 fbDosingStChart2(
	bWrite:= VIS.bDispencer1Dose, 
	udiCycleTime:= 5,
	lrAiData0:= VIS.lrDispencer2ActPos,
	lrAiData1:= VIS.lrDispencer12LifterActPos, 
	lrAiData2:= BOOL_TO_LREAL(P02_Dispencers.QbDispencer2SuckingValveActuator),
	lrAiData3:= BOOL_TO_LREAL(P02_Dispencers.QbDispencer2DosingValveActuator), 
	lrAiData4:= BOOL_TO_LREAL(P02_Dispencers.QbDispencer2DropCatcherValveActuator), 
	AiData=> VIS.AStAsChartDose2[0] );
	
fbDosingChart3(
	bWrite:= VIS.bDispencer3Dose, 
	nCycleTime:= 5,//nChartCycleTime, 
	lrData1:= VIS.lrDispencer3ActPos, 
	lrData2:= VIS.lrDispencer34LifterActPos, 
	bData3:= P02_Dispencers.QbDispencer3SuckingValveActuator, 
	bData4:= P02_Dispencers.QbDispencer3DosingValveActuator,
	bData5:= P02_Dispencers.QbDispencer3DropCatcherValveActuator,
	AsData=>VIS.AsChartDose3 );
	
 fbDosingStChart3(
	bWrite:= VIS.bDispencer1Dose, 
	udiCycleTime:= 5,
	lrAiData0:= VIS.lrDispencer3ActPos,
	lrAiData1:= VIS.lrDispencer34LifterActPos, 
	lrAiData2:= BOOL_TO_LREAL(P02_Dispencers.QbDispencer3SuckingValveActuator),
	lrAiData3:= BOOL_TO_LREAL(P02_Dispencers.QbDispencer3DosingValveActuator), 
	lrAiData4:= BOOL_TO_LREAL(P02_Dispencers.QbDispencer3DropCatcherValveActuator), 
	AiData=> VIS.AStAsChartDose3[0] );

fbDosingChart4(
	bWrite:= VIS.bDispencer4Dose, 
	nCycleTime:= 5,//nChartCycleTime, 
	lrData1:= VIS.lrDispencer4ActPos, 
	lrData2:= VIS.lrDispencer34LifterActPos, 
	bData3:= P02_Dispencers.QbDispencer4SuckingValveActuator, 
	bData4:= P02_Dispencers.QbDispencer4DosingValveActuator,
	bData5:= P02_Dispencers.QbDispencer4DropCatcherValveActuator,
	AsData=>VIS.AsChartDose4 );

fbDosingStChart4(
	bWrite:= VIS.bDispencer1Dose, 
	udiCycleTime:= 5,
	lrAiData0:= VIS.lrDispencer4ActPos,
	lrAiData1:= VIS.lrDispencer34LifterActPos, 
	lrAiData2:= BOOL_TO_LREAL(P02_Dispencers.QbDispencer4SuckingValveActuator),
	lrAiData3:= BOOL_TO_LREAL(P02_Dispencers.QbDispencer4DosingValveActuator), 
	lrAiData4:= BOOL_TO_LREAL(P02_Dispencers.QbDispencer4DropCatcherValveActuator), 
	AiData=> VIS.AStAsChartDose4[0] );
END_ACTION

ACTION aDropCatcher:
(**Uruchamianie ssawki tacek**)
P02_Dispencers.QbDispencerDropCatcherSuck;
IF (P00_PackML.fbPMLAuto.ePMLState = E_PMLState.ePMLState_EXECUTE OR P00_PackML.fbPMLModeManager.eModeStatus = E_PMLUnitMode.ePMLUnitMode_MANUAL) THEN
	fbDropCatcherSuck(T1:=T#5S , T0:=T#30S , Q=>P02_Dispencers.QbDispencerDropCatcherSuck);
	;
ELSE
	P02_Dispencers.QbDispencerDropCatcherSuck := FALSE;
END_IF

IF VIS.bDispencerManualDropCatcherSuck AND bManualMode THEN
	
	P02_Dispencers.QbDispencerDropCatcherSuck	:= TRUE;
END_IF
END_ACTION

ACTION aExSensor:


(** Czujnik Ex w zbiorniku **)

tonLowLevelExSensor(IN:=NOT IbTankLevelHighEX AND IbTankLevelLowEX AND NOT tonErrorExSensorDelay.Q AND bExEnable, PT:=T#1S);

IF tonLowLevelExSensor.Q THEN
	bTank1LevelExSensor:=TRUE;
ELSE
	bTank1LevelExSensor:=FALSE;
END_IF





//Błąd czujnika Ex
tonErrorExSensorDelay(IN:=IbTankLevelExError, PT:=T#5S);

IF tonErrorExSensorDelay.Q AND NOT TanksError.bError AND bExEnable AND bTank1SupplyPumpEnable THEN
	TanksError.bError:=TRUE;
	TanksError.bReset:=FALSE;
	TanksError.udiStationID:=78;
	TanksError.nErrorCode:=368;
	TanksError.sStationName:='Błąd systemu';
	TanksError.sErrorString:='Błąd czujnika poziomu Ex w zbiorniku. Sprawdz podłączenie lub stan separatora';
END_IF
END_ACTION

ACTION aLevelSensorCalibration:


(*
	bDialogBoxOn:BOOL;						(**)		// Wyświetlanie okienka komunikatów
	bDialogBoxText:STRING;					(**)		// Treść na oknie komunikatów
	bDialogBoxAck:BOOL;						(*t*)		// Potwierdzenie ogólne
	bDialogBoxCancelAck:BOOL;				(*t*)		// Wycofywanie procedury
	nDialogBoxType:UINT;								// Rodzaj okna, 0-nic, 1-tylko przysisk OK, 2 - tylko przycisk Anuluj, 3 - Przycisk OK i Anuluj
*)


(****Kalibracja czujnika nr 1 na pusto****)
tonTankLevelSensorCalibrationLight(IN:= nCalibrationDialog = 1 AND (VIS.bTank1LevelSensorCalibrationLight),PT:=T#10S);
tonTankLevelSensorCalibrationDark(IN:= nCalibrationDialog = 1 AND (VIS.bTank1LevelSensorCalibrationDark), PT:=T#5S);
IF VIS.bTank1LevelSensorCalibrationLight OR VIS.bTank1LevelSensorCalibrationDark THEN 		//Rozpoczaecie procedury kalibracji
	CASE nCalibrationDialog OF
		
		0: //Pytanie Czy na pewno
			VIS.nDialogBoxType	:=	3;									//Wyświetlanie przycisku OK i Anuluj
			IF VIS.bTank1LevelSensorCalibrationLight THEN
				VIS.bDialogBoxText	:=	'Want calibrate the level sensor to an empty tank? Immerse the sensor in the mass and remove it, simulating an empty tank.';
				VIS.sDialogBoxPicture	:= 'info';
			ELSIF VIS.bTank1LevelSensorCalibrationDark THEN
				VIS.bDialogBoxText	:=	'Should I calibrate the level sensor to a full tank? Immerse the sensor in the mass to simulate a full tank.';
				VIS.sDialogBoxPicture	:= 'info';
			END_IF
			VIS.bDialogBoxOn	:=	TRUE;
			IF VIS.bDialogBoxAck THEN
				VIS.bDialogBoxAck	:=	FALSE;		
				nCalibrationDialog:=nCalibrationDialog+1;
			ELSIF VIS.bDialogBoxCancelAck THEN
				VIS.bTank1LevelSensorCalibrationLight	:=	FALSE;
				VIS.bTank1LevelSensorCalibrationDark	:=	FALSE;

				//MAIN.aResetDialog();	
				nCalibrationDialog := 0;
			END_IF
			
		1: //Trwa kalibracja
			VIS.nDialogBoxType	:=	0;									//Bez przycisków
			
			IF VIS.bTank1LevelSensorCalibrationLight THEN
				QbTank1LevelSensorCalibration := NOT tonTankLevelSensorCalibrationLight.Q;	
				VIS.bDialogBoxText	:=	'Empty tank calibration in progress 1...';
				VIS.sDialogBoxPicture	:= '';
			END_IF
			IF VIS.bTank1LevelSensorCalibrationDark THEN
				QbTank1LevelSensorCalibration := NOT tonTankLevelSensorCalibrationDark.Q;	
				VIS.bDialogBoxText	:=	'Full tank calibration in progress 1...';
				VIS.sDialogBoxPicture	:= '';
			END_IF
			IF tonTankLevelSensorCalibrationLight.Q OR tonTankLevelSensorCalibrationDark.Q THEN
				nCalibrationDialog:=nCalibrationDialog+1;
			END_IF
			
		2: //Koniec kalibracji
			VIS.nDialogBoxType	:=	1;									//Potwierdz kalibracje
			VIS.bDialogBoxText	:=	'Calibration completed successfully';
			VIS.sDialogBoxPicture	:= 'ok';
			IF VIS.bTank1LevelSensorCalibrationLight OR VIS.bTank1LevelSensorCalibrationDark THEN
				bTank1LevelSensorCalibrated := TRUE;						//Zmienna presistent o kalibracji
			END_IF
			
			IF  VIS.bDialogBoxAck THEN
				VIS.bDialogBoxAck :=					FALSE;
				VIS.bTank1LevelSensorCalibrationLight	:=	FALSE;
				VIS.bTank1LevelSensorCalibrationDark	:=	FALSE;
				P00_Visualization.aResetDialog();
				nCalibrationDialog := 0;
			END_IF
			
	END_CASE
END_IF
END_ACTION

ACTION aLimits:

(*Zabezpieczenie nastaw dozowników*)
//Dozownika 1 i 2 (1 faza)
IF VIS.lrDispencer1DoseValveOpenTimeAccShow>0 			THEN 	VIS.lrDispencer1DoseValveOpenVolumeShow		:=0;		END_IF
IF VIS.lrDispencer1DoseValveCloseTimeDecShow>0 			THEN	VIS.lrDispencer1DoseValveCloseVolumeShow	:=0;		END_IF
IF VIS.bDispencer1DoseSuckingShow 						THEN	VIS.lrDispencer1DoseValveCloseVolumeShow	:=0;		END_IF
IF VIS.lrDispencer1SuckValveOpenTimeDelayShow>0 		THEN	VIS.lrDispencer1SuckValveOpenVolumeShow		:=0;		END_IF
IF VIS.lrDispencer1SuckValveCloseTimeDelayShow>0 		THEN	VIS.lrDispencer1SuckValveCloseVolumeShow	:=0;		END_IF
IF VIS.lrDispencer1Phase1VolumeShow > VIS.lrDispencer1DoseVolumeShow - VIS.lrDispencer1Phase2VolumeShow THEN	VIS.lrDispencer1Phase1VolumeShow	:= VIS.lrDispencer1DoseVolumeShow - VIS.lrDispencer1Phase2VolumeShow;END_IF
IF VIS.lrDispencer1Phase2VolumeShow > VIS.lrDispencer1DoseVolumeShow - VIS.lrDispencer1Phase1VolumeShow THEN	VIS.lrDispencer1Phase2VolumeShow 	:= VIS.lrDispencer1DoseVolumeShow - VIS.lrDispencer1Phase1VolumeShow;END_IF
IF VIS.lrDispencer1Phase2VolumeShow > VIS.lrDispencer1DoseVolumeShow 									THEN	VIS.lrDispencer1Phase1VolumeShow	:= 0;	VIS.lrDispencer1Phase2VolumeShow 	:= VIS.lrDispencer1DoseVolumeShow;END_IF

// Dozownika 3 i 4 (2 faza)
IF VIS.lrDispencer2DoseValveOpenTimeAccShow>0 			THEN	VIS.lrDispencer2DoseValveOpenVolumeShow		:=0;		END_IF
IF VIS.lrDispencer2DoseValveCloseTimeDecShow>0 			THEN	VIS.lrDispencer2DoseValveCloseVolumeShow	:=0;		END_IF
IF VIS.bDispencer2DoseSuckingShow 						THEN	VIS.lrDispencer2DoseValveCloseVolumeShow	:=0;		END_IF
IF VIS.lrDispencer2SuckValveOpenTimeDelayShow>0 		THEN	VIS.lrDispencer2SuckValveOpenVolumeShow		:=0;		END_IF
IF VIS.lrDispencer2SuckValveCloseTimeDelayShow>0 		THEN	VIS.lrDispencer2SuckValveCloseVolumeShow	:=0;		END_IF
IF VIS.lrDispencer2Phase1VolumeShow > VIS.lrDispencer2DoseVolumeShow - VIS.lrDispencer2Phase2VolumeShow THEN	VIS.lrDispencer2Phase1VolumeShow	:= VIS.lrDispencer2DoseVolumeShow - VIS.lrDispencer2Phase2VolumeShow;END_IF
IF VIS.lrDispencer2Phase2VolumeShow > VIS.lrDispencer2DoseVolumeShow - VIS.lrDispencer2Phase1VolumeShow THEN	VIS.lrDispencer2Phase2VolumeShow 	:= VIS.lrDispencer2DoseVolumeShow - VIS.lrDispencer2Phase1VolumeShow;END_IF
IF VIS.lrDispencer2Phase2VolumeShow > VIS.lrDispencer2DoseVolumeShow 									THEN	VIS.lrDispencer2Phase1VolumeShow	:= 0;	VIS.lrDispencer2Phase2VolumeShow 	:= VIS.lrDispencer2DoseVolumeShow;END_IF

IF lrDispencersLifterReadyPosition <1 					THEN	lrDispencersLifterReadyPosition			:=	270;													END_IF
IF 	VIS.lrDispencersLifterReadyPositionShow > 
	(P02_Dispencers.fbDispencer1.lrMaxPosition - 2)		THEN	VIS.lrDispencersLifterReadyPositionShow	:=	P02_Dispencers.fbDispencer1.lrMaxPosition - 2;			END_IF
	
	
IF 	VIS.lrFormsDragingLeftStartPosition		= 0		THEN	VIS.lrFormsDragingLeftStartPosition		:=	7;		END_IF;
IF 	VIS.lrFormsDragingLeftEndPosition		= 0		THEN	VIS.lrFormsDragingLeftEndPosition		:=	137;	END_IF;
IF 	VIS.lrFormsDragingRightStartPosition	= 0		THEN	VIS.lrFormsDragingRightStartPosition	:=	7.5;		END_IF;
IF 	VIS.lrFormsDragingRightEndPosition		= 0		THEN	VIS.lrFormsDragingRightEndPosition		:=	139;	END_IF;;
END_ACTION

ACTION aTankHeating:
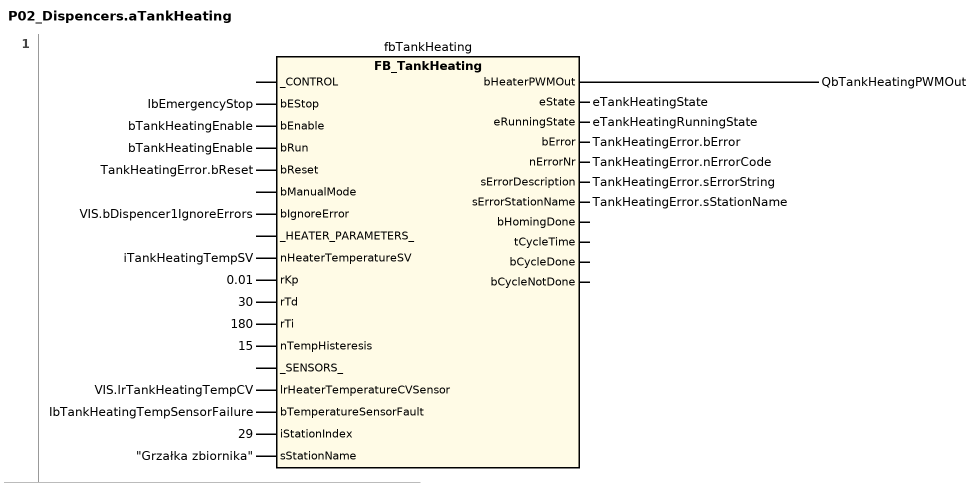
// NETWORK 1
fbTankHeating(
    bEStop := IbEmergencyStop,
    bEnable := bTankHeatingEnable,
    bRun := bTankHeatingEnable,
    bReset := TankHeatingError.bReset,
    bIgnoreError := VIS.bDispencer1IgnoreErrors,
    nHeaterTemperatureSV := iTankHeatingTempSV,
    rKp := 0.01,
    rTd := 30,
    rTi := 180,
    nTempHisteresis := 15,
    lrHeaterTemperatureCVSensor := VIS.lrTankHeatingTempCV,
    bTemperatureSensorFault := IbTankHeatingTempSensorFailure,
    iStationIndex := 29,
    sStationName := "Grzałka zbiornika",
    eState => eTankHeatingState,
    eRunningState => eTankHeatingRunningState,
    bError => TankHeatingError.bError,
    nErrorNr => TankHeatingError.nErrorCode,
    sErrorDescription => TankHeatingError.sErrorString,
    sErrorStationName => TankHeatingError.sStationName); // FB_TankHeating
QbTankHeatingPWMOut := fbTankHeating.bHeaterPWMOut;
END_ACTION

ACTION aTanks:
//Sterowanie Mieszadłem zbiornikowym
IF IbEmergencyStop (*AND IbFuseTankMixerEngineOK*) THEN
	QbTank1MixerStart:=(bTank1MixerEnable AND NOT bChangeover) OR (VIS.bTank1ManualMixer AND bManualMode);
ELSE
	QbTank1MixerStart:=FALSE;
	VIS.bTank1ManualMixer:=FALSE;
END_IF

//Sterowanie grzaniem zbiornika
//QbTank1HeaterOn:=IbEmergencyStopButton AND bTank1HeaterEnable OR (VIS.bManualTank1Heater AND bManualMode);

//Odwracanie sygnałów z czujników poziomu z receptur
bTank1LevelSignalInvert;									// Odwróć sygnał z czujnika zbiornika pierwszego
bTank2LevelSignalInvert;									// Odwróć sygnał z czujnika zbionirka drugiego
VIS.bTank1SupplyPumpEnableShow;
VIS.bTank2SupplyPumpEnableShow;
//Zmienne do poglądu zadziałania pomp od czujników
VIS.bHMITank1LevelSensorPumpOn;								// Sygnał z czujnika poziomu 1 załączający pompe 1 zależnie od ustawień (do podglądu sprawdzenia działania pompy bez jej załaczania)
VIS.bHMITank2LevelSensorPumpOn;								// Sygnał z czujnika poziomu 2 załączający pompe 2 zaleznie od ustawień (do podglądu sprawdzenia działania pompy bez jej załaczania)

//Odwracanie sygnałów z czujników poziomu
IF NOT bTank1LevelSignalInvert THEN
	bTank1LevelLow					:=	IbTank1LevelLow OR bTank1LevelLowConductiveSensor OR bTank1LevelExSensor; 	
	VIS.bHMITank1LevelSensorPumpOn	:=	IbTank1LevelLow OR bTank1LevelLowConductiveSensor OR bTank1LevelExSensor; 	
ELSE
	bTank1LevelLow					:=	NOT IbTank1LevelLow;
	VIS.bHMITank1LevelSensorPumpOn	:=	NOT IbTank1LevelLow;
END_IF
IF NOT bTank2LevelSignalInvert THEN
	bTank2LevelLow					:=	IbTank2LevelLow OR bTank2LevelLowConductiveSensor;
	VIS.bHMITank2LevelSensorPumpOn	:=	IbTank2LevelLow OR bTank2LevelLowConductiveSensor;
ELSE
	bTank2LevelLow					:=	NOT IbTank2LevelLow;	
	VIS.bHMITank2LevelSensorPumpOn	:=	NOT IbTank2LevelLow;
END_IF

// Mycie CIP

IF bCIP THEN
	tonTank1LevelSensor(IN:= bTank1LevelLow,PT:=T#15S);
ELSE
	IF VIS.lrDispencer1DoseVolumeShow > 450 THEN
		tonTank1LevelSensor(IN:= bTank1LevelLow,PT:=T#500MS);
	ELSE
		tonTank1LevelSensor(IN:= bTank1LevelLow,PT:=T#5S);		
	END_IF
END_IF
	
//Sterowanie pompą podającą nr 1
tofTank1LevelSensor(IN:= bTank1LevelLow,PT:=T#0S);

IF IbEmergencyStop AND (tofTank1LevelSensor.Q OR  tonTank1LevelSensor.Q) AND NOT GVL.SensorAcetoneError.bError AND NOT bHomingDialog THEN  // dodany sygnał od czujnika acetonu
	QbTank1PumpStart:=(bTank1SupplyPumpEnable AND NOT bChangeover) OR (VIS.bTank1ManualSupplyPump AND bManualMode);
ELSE
	QbTank1PumpStart:=FALSE;
END_IF

//Sterowanie pompą podającą nr 2
tofTank2LevelSensor(IN:= bTank2LevelLow,PT:=T#0S);
tonTank2LevelSensor(IN:= bTank2LevelLow,PT:=T#5S);
IF IbEmergencyStop AND (tofTank2LevelSensor.Q OR tonTank2LevelSensor.Q) AND NOT bHomingDialog THEN  // dodany sygnał od czujnika acetonu THEN
	QbTank2PumpStart:=(bTank2SupplyPumpEnable AND NOT bChangeover) OR (VIS.bTank2ManualSupplyPump AND bManualMode);
ELSE
	QbTank2PumpStart:=FALSE;
END_IF

//ERROR HANDLING
// Alarm_0100	100	Error	Zbiornik 1 | Brak masy w leju
// Alarm_0101	101	Error	Zbiornik 2 | Brak masy w leju
// Alarm_0102	102	Error	Mixer | Wyłączone zabezpieczenie przy próbie uruchomienia
// Alarm_0103	103	Error	Pompa 1 | Przepalony bezpiecznik - sprawdź połączenie i wymień
// Alarm_0104	104	Error	Pompa 2 | Przepalony bezpiecznik - sprawdź połączenie i wymień

IF bAlarmInit THEN
    bAlarmInit := FALSE; 
	fbSourceInfo.Clear();
	fbSourceInfo.sName:='Błąd systemu';//sStationName;//'Machine';
	fbSourceInfo.nId:=78;//udiStationID;//2700;
	// Alarm_0100	100	Error	Zbiornik 1 | Brak masy w leju
    arfbAlarm[0].CreateEx(stEventEntry := TC_EVENTS.AlarmClass.Alarm_0100, bWithConfirmation:= FALSE,  ipSourceInfo:= fbSourceInfo); 
	// Alarm_0101	101	Error	Zbiornik 2 | Brak masy w leju
	arfbAlarm[1].CreateEx(stEventEntry := TC_EVENTS.AlarmClass.Alarm_0101, bWithConfirmation:= FALSE,  ipSourceInfo:= fbSourceInfo); 
	// Alarm_0102	102	Error	Mixer | Wyłączone zabezpieczenie przy próbie uruchomienia
	arfbAlarm[2].CreateEx(stEventEntry := TC_EVENTS.AlarmClass.Alarm_0102, bWithConfirmation:= FALSE,  ipSourceInfo:= fbSourceInfo); 
	// Alarm_0103	103	Error	Pompa 1 | Przepalony bezpiecznik - sprawdź połączenie i wymień
	arfbAlarm[3].CreateEx(stEventEntry := TC_EVENTS.AlarmClass.Alarm_0103, bWithConfirmation:= FALSE,  ipSourceInfo:= fbSourceInfo); 
	// Alarm_0104	104	Error	Pompa 2 | Przepalony bezpiecznik - sprawdź połączenie i wymień
	arfbAlarm[4].CreateEx(stEventEntry := TC_EVENTS.AlarmClass.Alarm_0104, bWithConfirmation:= FALSE,  ipSourceInfo:= fbSourceInfo); 
END_IF


// Alarm_0100	100	Error	Zbiornik 1 | Brak masy w leju
//BŁĄD 72- Brak masy w leju	zbiorniku 1
//tonTank1EmptyAlarm(IN:=bTank1LevelLow AND (eMachineState=E_MachineState.eCycleOn OR eMachineState=E_MachineState.eCycleStarting OR eMachineState = E_MachineState.eConfectionEnd),PT:=T#25S);
//Opcja z liczeniem ilości doz
IF bTank1SupplyPumpEnable AND (tonTank1EmptyAlarm.Q OR nDose1CounterWhenLowLevel>=nDoseCounter1) AND NOT VIS.bTanksIgnoreError THEN
	IF NOT arfbAlarm[0].bActive THEN
			arfbAlarm[0].Raise(nTimeStamp:=0);
		END_IF
	ELSE	
		IF  arfbAlarm[0].bActive AND TanksError.bReset THEN
			arfbAlarm[0].Clear(nTimeStamp:=0, bResetConfirmation:= FALSE);
	END_IF	
// 	TanksError.bError:=TRUE;
// 	TanksError.bReset:=FALSE;
// 	TanksError.udiStationID:=78;
// 	TanksError.nErrorCode:=72;
// 	TanksError.sStationName:='Błąd systemu';
// 	TanksError.sErrorString:='Zbiornik 1 | Brak masy w leju';
END_IF
// Alarm_0101	101	Error	Zbiornik 2 | Brak masy w leju
//BŁĄD 73- Brak masy w leju	zbiorniku 2																	
//tonTank2EmptyAlarm(IN:=bTank2LevelLow AND (eMachineState=E_MachineState.eCycleOn OR eMachineState=E_MachineState.eCycleStarting OR eMachineState = E_MachineState.eConfectionEnd),PT:=T#25S);
//Opcja z liczeniem ilości doz
//tonTank2EmptyAlarm(IN:=(bTank2LevelLow OR nDose2CounterWhenLowLevel>=nDoseCounter2)	AND (P00_PackML.fbPMLAuto.ePMLState = E_PMLState.ePMLState_EXECUTE OR P00_PackML.fbPMLAuto.ePMLState = E_PMLState.ePMLState_STARTING),PT:=T#25S);
IF bTank2SupplyPumpEnable AND (tonTank2EmptyAlarm.Q OR nDose2CounterWhenLowLevel>=nDoseCounter1) AND NOT VIS.bTanksIgnoreError THEN
		IF NOT arfbAlarm[1].bActive THEN
			arfbAlarm[1].Raise(nTimeStamp:=0);
		END_IF
	ELSE	
		IF  arfbAlarm[1].bActive AND TanksError.bReset THEN
			arfbAlarm[1].Clear(nTimeStamp:=0, bResetConfirmation:= FALSE);
	END_IF
// 	TanksError.bError:=TRUE;
// 	TanksError.bReset:=FALSE;
// 	TanksError.udiStationID:=78;
// 	TanksError.nErrorCode:=73;
// 	TanksError.sStationName:='Błąd systemu';
// 	TanksError.sErrorString:='Zbiornik 2 | Brak masy w leju';
END_IF
// Alarm_0102	102	Error	Mixer | Wyłączone zabezpieczenie przy próbie uruchomienia
//BŁĄD 74- Błąd zabezpieczenia mieszadła podczas właczenia zasilania jednego
tonMixerNotWorking(IN:=NOT IbFuseTankMixerEngineOK AND QbTank1MixerStart, PT:=T#3S);
IF tonMixerNotWorking.Q THEN
		IF NOT arfbAlarm[2].bActive THEN
			arfbAlarm[2].Raise(nTimeStamp:=0);
		END_IF
	ELSE	
		IF  arfbAlarm[2].bActive AND TanksError.bReset THEN
			arfbAlarm[2].Clear(nTimeStamp:=0, bResetConfirmation:= FALSE);
	END_IF
// 	TanksError.bError:=TRUE;
// 	TanksError.bReset:=FALSE;
// 	TanksError.udiStationID:=78;
// 	TanksError.nErrorCode:=74;
// 	TanksError.sStationName:='Błąd systemu';
// 	TanksError.sErrorString:='Mixer | Wyłączone zabezpieczenie przy próbie uruchomienia';
END_IF
// Alarm_0103	103	Error	Pompa 1 | Przepalony bezpiecznik - sprawdź połączenie i wymień
//BŁĄD 75 - Przepalony bezpiecznik pompy 1 
tonTank1PumpFuseOK(IN:= QbTank1PumpStart AND NOT IbTank1PumpFuseOK, PT:= T#1S);
IF tonTank1PumpFuseOK.Q  THEN
		IF NOT arfbAlarm[3].bActive THEN
			arfbAlarm[3].Raise(nTimeStamp:=0);
		END_IF
	ELSE	
		IF  arfbAlarm[3].bActive AND TanksError.bReset THEN
			arfbAlarm[3].Clear(nTimeStamp:=0, bResetConfirmation:= FALSE);
	END_IF
// 	TanksError.bError:=TRUE;
// 	TanksError.bReset:=FALSE;
// 	TanksError.udiStationID:=78;
// 	TanksError.nErrorCode:=75;
// 	TanksError.sStationName:='Błąd systemu';
// 	TanksError.sErrorString:='Pompa 1 | Przepalony bezpiecznik - sprawdź połączenie i wymień';
END_IF
// Alarm_0104	104	Error	Pompa 2 | Przepalony bezpiecznik - sprawdź połączenie i wymień
//BŁĄD 76- Przepalony bezpiecznik pompy 2 
tonTank2PumpFuseOK(IN:= QbTank2PumpStart AND NOT IbTank2PumpFuseOK, PT:= T#1S);
IF tonTank2PumpFuseOK.Q THEN
		IF NOT arfbAlarm[4].bActive THEN
			arfbAlarm[4].Raise(nTimeStamp:=0);
		END_IF
	ELSE	
		IF  arfbAlarm[4].bActive AND TanksError.bReset THEN
			arfbAlarm[4].Clear(nTimeStamp:=0, bResetConfirmation:= FALSE);
	END_IF
// 	TanksError.bError:=TRUE;
// 	TanksError.bReset:=FALSE;
// 	TanksError.udiStationID:=78;
// 	TanksError.nErrorCode:=76;
// 	TanksError.sStationName:='Błąd systemu';
// 	TanksError.sErrorString:='Pompa 2 | Przepalony bezpiecznik - sprawdź połączenie i wymień';
END_IF



//BŁĄD 21- zaklejenie czujnika w zbiorniku	
rtDispencer1DoseDone(CLK:=P02_Dispencers.fbDispencer1.bCycleDone,Q=>);
rtDispencer2DoseDone(CLK:=P02_Dispencers.fbDispencer2.bCycleDone,Q=>);

IF bTank1LevelLow THEN
	nDose1Counter:=0;
ELSIF rtDispencer1DoseDone.Q THEN
	nDose1Counter:=nDose1Counter+1;
END_IF

IF bTank2LevelLow THEN
	nDose2Counter:=0;
ELSIF rtDispencer2DoseDone.Q THEN
	nDose2Counter:=nDose2Counter+1;
END_IF

IF rtDispencer1DoseDone.Q  AND bTank1LevelLow THEN
	nDose1CounterWhenLowLevel := nDose1CounterWhenLowLevel	+	1;
END_IF
IF rtDispencer2DoseDone.Q AND bTank2LevelLow THEN
	nDose2CounterWhenLowLevel := nDose2CounterWhenLowLevel	+	1;
END_IF
IF NOT bTank1LevelLow THEN
	nDose1CounterWhenLowLevel := 0;
END_IF
IF NOT bTank2LevelLow THEN
	nDose2CounterWhenLowLevel := 0;
END_IF

(*Obliczanie wartości liczby dozy po których jest alarm zależnie od dozy*)

IF NOT bDosingTwoPhases THEN
	IF lrDispencer1DoseVolume > 0 AND lrDispencer1DoseVolume < 300 THEN //Zawsze błąd po 2 litrach na jeden dozownik czyli 4 litry
		nDoseCounter1 := LREAL_TO_INT( 827 * EXPT(lrDispencer1DoseVolume,-0.959));
		//nDoseCounter1 := LREAL_TO_INT( 2467.3 * EXPT(lrDispencer1DoseVolume,-1.082));		
	ELSIF 	lrDispencer1DoseVolume > 600 THEN
		nDoseCounter1 := 4;
	ELSIF 	lrDispencer1DoseVolume > 450 THEN
		nDoseCounter1 := 8;
	ELSIF 	lrDispencer1DoseVolume > 300 THEN
		nDoseCounter1 := 13;		
	ELSE
		nDoseCounter1 := 25 ;
	END_IF
ELSE
	IF lrDispencer1DoseVolume > 0 THEN //Zawsze błąd po 2 litrach na jeden dozownik czyli 4 litry
		nDoseCounter1 := LREAL_TO_INT( 827 * EXPT(lrDispencer1DoseVolume,-0.959));
		//nDoseCounter1 := LREAL_TO_INT( 2467.3 * EXPT(lrDispencer1DoseVolume,-1.082));		
	ELSE
		nDoseCounter1 := 25 ;
	END_IF
	IF lrDispencer2DoseVolume > 0 THEN //Zawsze błąd po 2 litrach na jeden dozownik czyli 4 litry
		nDoseCounter2 := LREAL_TO_INT( 827 * EXPT(lrDispencer2DoseVolume,-0.959));
		//nDoseCounter2 := LREAL_TO_INT( 2467.3 * EXPT(lrDispencer2DoseVolume,-1.082));		
	ELSE
		nDoseCounter2 := 25 ;
	END_IF
END_IF
IF nDoseCounter1 < 3 THEN	nDoseCounter1 := 3;END_IF
IF nDoseCounter2 < 3 THEN	nDoseCounter2 := 3;END_IF

(*IF bTank1SupplyPumpEnable AND nDose1Counter>nDoseCounter1 AND NOT TanksError.bError AND NOT VIS.bTanksIgnoreError THEN
	TanksError.bError:=TRUE;
	TanksError.bReset:=FALSE;
	TanksError.nErrorCode:=22;
	TanksError.sStationName:='Zbiornik 1';
	TanksError.sErrorString:='Zaklejony czujnik w zbiorniku';
END_IF*)

(*IF bTank2SupplyPumpEnable AND nDose2Counter>nDoseCounter2 AND NOT TanksError.bError AND NOT VIS.bTanksIgnoreError THEN
	TanksError.bError:=TRUE;
	TanksError.bReset:=FALSE;
	TanksError.nErrorCode:=23;
	TanksError.sStationName:='Zbiornik 2';
	TanksError.sErrorString:='Zaklejony czujnik w zbiorniku';
END_IF*)

IF TanksError.bReset THEN
	nDose1CounterWhenLowLevel := 0;
	nDose2CounterWhenLowLevel := 0;
	nDose1Counter := 0;
	nDose2Counter := 0;
//	TanksError.bError:=FALSE;
//	TanksError.bReset:=FALSE;
//	TanksError.nErrorCode:=0;
//	TanksError.sStationName:='';
//	TanksError.sErrorString:='';
END_IF

(*Wyświetlanie błedu na wyjściu*)
TanksError.bError							:= FALSE;
FOR nAlarmNumerator := 0 TO 19 DO
	TanksError.bError						:= TanksError.bError OR arfbAlarm[nAlarmNumerator].bActive;
END_FOR

(***Ciśnienie w zbiornikach****)
P02_Dispencers.QbTank1Pressure:=(bTank1PressureEnable AND NOT bChangeover) OR (VIS.bTank1ManualPressure AND bManualMode);

(***WYŁĄCZANIE JEZELI NIE SA W TRYBIE SERWISOWYM***)
IF NOT bManualMode THEN
	VIS.bTank1ManualSupplyPump := FALSE;
	VIS.bTank2ManualSupplyPump := FALSE;
	VIS.bTank1ManualPressure := FALSE;
	VIS.bTank1ManualMixer := FALSE;
END_IF
END_ACTION

ACTION aTanksRainbowMode:
VIS.bTankRainbowModeShow;
bTankRainbowMode;

VIS.bHMITank3LevelSensorPumpOn;	
VIS.iTank3LevelSensorValue;		
VIS.bHMITank4LevelSensorPumpOn;	
VIS.iTank4LevelSensorValue;		

VIS.uTank1LevelSetpointShow;
VIS.uTank1LevelSetpointShow;
END_ACTION

ACTION aTankWarning:

(****Ostrzezenia***)
//Niski poziom w zbiorniku 1
tonTank1LevelWarning (IN:=	VIS.iTank1LevelSensorValue < 10 AND 
							P00_PackML.fbPMLAuto.ePMLState =	Tc3_PackML.E_PMLState.ePMLState_EXECUTE
					, PT:=T#3S);

IF tonTank1LevelWarning.Q AND NOT TanksWarning[0].bWarning THEN
	TanksWarning[0].bWarning									:=TRUE;
	TanksWarning[0].udiWarningCode								:=25;
	TanksWarning[0].sDescription								:= 'Zbiornik 1 | Niski poziom w zbiorniku';
ELSIF NOT tonTank1LevelWarning.Q AND TanksWarning[0].bAcknowledge THEN
	TanksWarning[0].bWarning									:=FALSE;
	TanksWarning[0].bAcknowledge								:=FALSE;
	VIS.uliWarningAcknowledge.0 								:=FALSE;
ELSIF TanksWarning[0].bAcknowledge THEN
	TanksWarning[0].bAcknowledge								:=TRUE;
END_IF

//Niski poziom w zbiorniku 2
tonTank1LevelWarning (IN:=	VIS.iTank2LevelSensorValue < 10 AND bDosingTwoPhases AND 
							P00_PackML.fbPMLAuto.ePMLState =	Tc3_PackML.E_PMLState.ePMLState_EXECUTE
					, PT:=T#3S);

IF tonTank1LevelWarning.Q AND NOT TanksWarning[1].bWarning THEN
	TanksWarning[1].bWarning									:=TRUE;
	TanksWarning[1].udiWarningCode								:=26;
	TanksWarning[1].sDescription								:= 'Zbiornik 2 | Niski poziom w zbiorniku';
ELSIF NOT tonTank1LevelWarning.Q AND TanksWarning[1].bAcknowledge THEN
	TanksWarning[1].bWarning									:=FALSE;
	TanksWarning[1].bAcknowledge								:=FALSE;
	VIS.uliWarningAcknowledge.1 								:=FALSE;
ELSIF TanksWarning[1].bAcknowledge THEN
	TanksWarning[1].bAcknowledge								:=TRUE;
END_IF
END_ACTION

ACTION aTDRMassSensor:
(*
Nazwa:			aTDRMassSensor
Opis:			Czujnik poziomu z prętem SICK 
Wersja:			v1.0
Data:			2021-05-17
Autor:			DP,MP
Urzadzenia:		Sick LFP
Konfiguracja:	
Info:
- przypisać zmienna od diagnostyki do blędów IO-LINK, żeby po wypięciu czujnika nie zaczeła pompowac pompa
- Ustawienia czujnika:
Parameter menu>PARAMETERS	>DspVAL-Distan
							>FIlter 400ms
				>EXPERT		>Mode Pulse
							>MeasMd HiAcc
							>MaxCol	10cm/s
				>Pulse		>TrsHld	50 NAJWAZNIEJSZE
							>CalRng 6005	
							>MaskZn 0
							>MaskTr 50
				>Probe		>Lenght 305
							>CblLen 1000
							>Type Rod
Kalibracja na pustym zbiorniku
SigQua musi byc powyżej 40 jeżeli wykrywa mase
Jeżeli nie wykrywa masy lub coś jest nie tak nalezy zwiększyć TrsHld
Za każdą zmianą trzeba kalibrowac czujnik
- Pompowanie zawsze do 150mm czujnika

*)


(*Przypisane na stałe*)
(*IF VIS.bTank1LevelSensorLow THEN // Poziom zależnie od nastaw
	VIS.uTank1LevelSetpointShow:=1;
ELSIF VIS.bTank1LevelSensorHigh THEN // Poziom zależnie od nastaw
	VIS.uTank1LevelSetpointShow:=120; //bylo 150
ELSE
	VIS.uTank1LevelSetpointShow:=140; //bylo 120
END_IF*)

IF VIS.uTank1LevelSetpointShow > 201 THEN
	VIS.uTank1LevelSetpointShow := 100;
END_IF



(**************************** ZBIORNIK 1***********************************************************)
(*Przypisanie zmiennych wizualiazji do zmiennych wewnetrznych programu*)
                     
iTank1Sensor1ValueTemp.0		:= 			IusiTank1SensorValue0.7		;
iTank1Sensor1ValueTemp.1		:= 			IusiTank1SensorValue0.6		;
iTank1Sensor1ValueTemp.2		:= 			IusiTank1SensorValue0.5		;
iTank1Sensor1ValueTemp.3		:= 			IusiTank1SensorValue0.4		;
iTank1Sensor1ValueTemp.4		:= 			IusiTank1SensorValue0.3		;
iTank1Sensor1ValueTemp.5		:= 			IusiTank1SensorValue0.2		;
iTank1Sensor1ValueTemp.6		:= 			IusiTank1SensorValue0.1		;
iTank1Sensor1ValueTemp.7		:= 			IusiTank1SensorValue0.0		;                                					
iTank1Sensor1ValueTemp.8		:= 			IusiTank1SensorValue1.7		;
iTank1Sensor1ValueTemp.9		:= 			IusiTank1SensorValue1.6		;
iTank1Sensor1ValueTemp.10		:= 			IusiTank1SensorValue1.5		;
iTank1Sensor1ValueTemp.11		:= 			IusiTank1SensorValue1.4		;
iTank1Sensor1ValueTemp.12		:= 			IusiTank1SensorValue1.3		;
iTank1Sensor1ValueTemp.13		:= 			IusiTank1SensorValue1.2		;
													
iTank1Sensor1Value.0			:=			iTank1Sensor1ValueTemp.13	;
iTank1Sensor1Value.1			:=			iTank1Sensor1ValueTemp.12	;													
iTank1Sensor1Value.2			:=			iTank1Sensor1ValueTemp.11	;													
iTank1Sensor1Value.3			:=			iTank1Sensor1ValueTemp.10	;													
iTank1Sensor1Value.4			:=			iTank1Sensor1ValueTemp.9	;													
iTank1Sensor1Value.5			:=			iTank1Sensor1ValueTemp.8	;													
iTank1Sensor1Value.6			:=			iTank1Sensor1ValueTemp.7	;													
iTank1Sensor1Value.7			:=			iTank1Sensor1ValueTemp.6	;													
iTank1Sensor1Value.8			:=			iTank1Sensor1ValueTemp.5	;													
iTank1Sensor1Value.9			:=			iTank1Sensor1ValueTemp.4	;													
iTank1Sensor1Value.10			:=			iTank1Sensor1ValueTemp.3	;													
iTank1Sensor1Value.11			:=			iTank1Sensor1ValueTemp.2	;													
iTank1Sensor1Value.12			:=			iTank1Sensor1ValueTemp.1	;													
iTank1Sensor1Value.13			:=			iTank1Sensor1ValueTemp.0	;													

(***Skalownaie wartości zadanej na 1-100%************)
(*Filtrowanie sygnału jeżeli włączony jest CIP*)
IF bCIP THEN
	fbFilterExiTank1Sensor1Value(
				rIn:=				INT_TO_REAL(iTank1Sensor1Value), 
				tTimeConstant:= 	T#50MS, 
				rOut=>				);
	VIS.iTank1LevelSensorValue := REAL_TO_INT(fbFilterExiTank1Sensor1Value.rOut);	
ELSE
//	VIS.iTank1LevelSensorValue := iTank1Sensor1Value;
END_IF
(****Koniec skalownaie wartości zadanej na 1-100%****)
																																												
bTank1SensorDiagnosis										:= NOT P00_PneumaticValves.fbiTank1LevelSensorValue.bError;

IF uTank1LevelSetpoint>290 THEN
	uTank1LevelSetpoint:=290;//Zabezpieczenie przed zbyt wielka nastawą
END_IF

//ZAŁĄCZANIE POMPY OD ZADANEJ WARTOŚCI
IF VIS.lrDispencer1DoseVolumeShow > 450 THEN
	tonTank1LevelLowConductiveSensor( IN:=VIS.iTank1LevelSensorValue < UINT_TO_INT(uTank1LevelSetpoint) AND bTank1SensorDiagnosis AND NOT bExEnable, PT:=T#1S);
ELSE
	tonTank1LevelLowConductiveSensor( IN:=VIS.iTank1LevelSensorValue < UINT_TO_INT(uTank1LevelSetpoint) AND bTank1SensorDiagnosis AND NOT bExEnable, PT:=T#10S);	
END_IF


IF tonTank1LevelLowConductiveSensor.Q THEN
	bTank1LevelLowConductiveSensor := TRUE;
ELSE
	bTank1LevelLowConductiveSensor := FALSE;
END_IF
(****************************KONIEC ZBIORNIK 1***********************************************************)

(*Przypisane na stałe*)

//VIS.uTank2LevelSetpointShow:=75; // bylo 120
IF VIS.uTank2LevelSetpointShow > 201 THEN
	VIS.uTank2LevelSetpointShow := 100;
END_IF

(**************************** ZBIORNIK 2***********************************************************)
                     
	iTank2Sensor1ValueTemp.0		:= 			IusiTank2SensorValue0.7		;
	iTank2Sensor1ValueTemp.1		:= 			IusiTank2SensorValue0.6		;
	iTank2Sensor1ValueTemp.2		:= 			IusiTank2SensorValue0.5		;
	iTank2Sensor1ValueTemp.3		:= 			IusiTank2SensorValue0.4		;
	iTank2Sensor1ValueTemp.4		:= 			IusiTank2SensorValue0.3		;
	iTank2Sensor1ValueTemp.5		:= 			IusiTank2SensorValue0.2		;
	iTank2Sensor1ValueTemp.6		:= 			IusiTank2SensorValue0.1		;
	iTank2Sensor1ValueTemp.7		:= 			IusiTank2SensorValue0.0		;                                					
	iTank2Sensor1ValueTemp.8		:= 			IusiTank2SensorValue1.7		;
	iTank2Sensor1ValueTemp.9		:= 			IusiTank2SensorValue1.6		;
	iTank2Sensor1ValueTemp.10		:= 			IusiTank2SensorValue1.5		;
	iTank2Sensor1ValueTemp.11		:= 			IusiTank2SensorValue1.4		;
	iTank2Sensor1ValueTemp.12		:= 			IusiTank2SensorValue1.3		;
	iTank2Sensor1ValueTemp.13		:= 			IusiTank2SensorValue1.2		;
														
	iTank2Sensor1Value.0			:=			iTank2Sensor1ValueTemp.13	;
	iTank2Sensor1Value.1			:=			iTank2Sensor1ValueTemp.12	;													
	iTank2Sensor1Value.2			:=			iTank2Sensor1ValueTemp.11	;													
	iTank2Sensor1Value.3			:=			iTank2Sensor1ValueTemp.10	;													
	iTank2Sensor1Value.4			:=			iTank2Sensor1ValueTemp.9	;													
	iTank2Sensor1Value.5			:=			iTank2Sensor1ValueTemp.8	;													
	iTank2Sensor1Value.6			:=			iTank2Sensor1ValueTemp.7	;													
	iTank2Sensor1Value.7			:=			iTank2Sensor1ValueTemp.6	;													
	iTank2Sensor1Value.8			:=			iTank2Sensor1ValueTemp.5	;													
	iTank2Sensor1Value.9			:=			iTank2Sensor1ValueTemp.4	;													
	iTank2Sensor1Value.10			:=			iTank2Sensor1ValueTemp.3	;													
	iTank2Sensor1Value.11			:=			iTank2Sensor1ValueTemp.2	;													
	iTank2Sensor1Value.12			:=			iTank2Sensor1ValueTemp.1	;													
	iTank2Sensor1Value.13			:=			iTank2Sensor1ValueTemp.0	;													
	     
	(****Koniec skalownaie wartości zadanej na 1-100%****)
																																													
	bTank2SensorDiagnosis										:= NOT P00_PneumaticValves.fbiTank2LevelSensorValue.bError;

VIS.iTank2LevelSensorValue := iTank2Sensor1Value;	
	//ZAŁĄCZANIE POMPY OD ZADANEJ WARTOŚCI
//ZAŁĄCZANIE POMPY OD ZADANEJ WARTOŚCI
tonTank2LevelLowConductiveSensor( IN:=VIS.iTank2LevelSensorValue < UINT_TO_INT(uTank2LevelSetpoint) AND bTank2SensorDiagnosis AND NOT bExEnable, PT:=T#10S);
IF tonTank2LevelLowConductiveSensor.Q THEN
	bTank2LevelLowConductiveSensor := TRUE;
ELSE
	bTank2LevelLowConductiveSensor := FALSE;
END_IF
(****************************KONIEC ZBIORNIK 2***********************************************************)
END_ACTION

END_PROGRAM

// ---- POUs/FB/FB_ServoDispencerServoLifter.TcPOU
(*
Nazwa:			FB_ServoDispencerFestoLifter
Opis:			Dozownik 
Wersja:			v0.67
Data:			2025-09-04
Autor:			DP
Urzadzenia:		Serwo dozowania, silniki krokowe podnoszenia FESTO, zawor ssania-dozowania
Konfiguracja:	
Zmiany:
- 20250904 [DP] EventLog-do sprawdzenia, 1 spr->wywołać błędy 
- 20250627 [DP] SoftReset False
- 20250626 [DP] GoingUp
- 20250303 [DP] limit dozy
- 20241217 [DP] Drop false jezeli pozycja ready < tacki
- 20241203 [AS] Dodana obsluga błędów od bloków MC osi Lifter oraz Dispencer, zerowanie "iCaseGoingUp" w Runnig --> ready
- 20241108 [DP] DoseAcc
- 20241025 [DP] Zmiana tasku i blad
- 20241017 [DP] Zmiana CatchSV na StopDose+5
- 20240612 [DP] Zmiana CatchSV usunięcie -5
- 20240322 [DP] Stan tacki do bledu
- 20240318 [DP] Czas estop błąd
- 20240311 [DP] Max lift vel.
- 20240205 [DP] Zmianiony PackML
- 20231215 [DP] DoseSucking jak delay >0, zla pozycja, tonError2 bo 1 uruch. er.
- 20230517 [DP] Zmiana Delay i Limitów, z XTS Z
- 20230303 [DP] Poprawiony SuckingValve w Manual
Info: 
-Zmieniono zachowanie po HomingDone
-Dodano opisy błędów serwa
-Zmiana zachowania tacki po wylaczeniu enable
-Dodano HomingNeeded
-Ulepszono przerywanie dozowania
-Enable Festo, dopiero jak nie ma warningu i jest zasilanie
-falsowanie enable festo na koncu
-Dodanie wysokosci tacki okapowej
*)
FUNCTION_BLOCK FB_ServoDispencerServoLifter
VAR_INPUT
    bEnable              : BOOL;          //Zezwolenie na pracę
	bChangeover			 : BOOL;	
    bEStop               : BOOL;          //Stop Awaryjny Całość
    bEStopButtonsAndDoors: BOOL;          //Stop Awaryjny	
	bInLimitSwitchSensor : BOOL; 		  //Krańcówka dosunięcia stacji
    bRun                 : BOOL;          //Rozkaz dozowania 
    bHoming              : BOOL;          //Zezwolenie na wykonanie bazowania (głównie po wykonanych mechanicznych zmianach)
    bHeightSet           : BOOL;          //Zezwolenie na wykonanie bazowania (głównie po wykonanych mechanicznych zmianach)
    bIgnoreError         : BOOL;          //Ignorowania błędów cyklu pracy
    bReset               : BOOL;          //Reset błędu, jeśli w stanie "eError"
    eGlobalState         : E_PMLState; 	//Stan ogólny maszyny, tylko do błędu
    bCatchEnable         : BOOL;          //Zezwolenie na pracę chwytaka, tylko do błędu
    lrDoseVolume         : LREAL;         //Ilość do wydozowania w [ml]
    bDispencerWithLifter : BOOL;          //OPCJA Dozownik z podnośnikiem
    bMultiMasterSyncIn   : BOOL;          //OPCJA Synchronizacja gotowsci innych dozowników // Jezeli ma działać niezależnie to ma być cały czas na TRUE
    bLiftSynchroPh1      : BOOL;          //Synchronizacja podnośnika z Dozownikiem w fazie 1
    bLiftSynchroPh2      : BOOL;          //Synchronizacha podnośnika z Dozownikiem w fazie 2
    bLiftSynchroPh3      : BOOL;          //Synchronizacja podnośnika z Dozownikiem w fazie 3

    //Parametryzacja dozownika (można wpisać na stałe)
	lrMaxDispencerVelocity		: LREAL;		//Max prędkość tłoka
    lrMaxPosition      			: LREAL; 		//Pozycja maksymalna podnośnika
    lrMinPosition      			: LREAL; 		//Pozycja minimalna podnośnika
    lrRatedDose        			: LREAL; 		//Znamionowa pojemność dozownika [ml];
    lrCylinderDiameter 			: LREAL;		//Średnica cylindra dozownika [mm]
	lrDropCatcherOpenDistance	: LREAL:=10;	//Różnica od aktualnej wysokości chwytaka przy której ma się otworzyć tacka (Domyślnie 10)

    //Informacje z czujników
    bSuckingValveOpenedSensor : BOOL;  //Czujnik otwarcia zaworu ssacego
    bSuckingValveClosedSensor : BOOL;  //Czujnik zamkmnięcia zaworu ssącego
    bDosingValveOpenedSensor  : BOOL;  //Czujnik otwarcia zaworu tłoczącego (iglicy)
    bDosingValveClosedSensor  : BOOL;  //Czujnik zamknięcia zaworu tłoczącego (iglicy) (tylko ten ma znaczenie w cyklu)
    bDropCatcherBackSensor    : BOOL;  //Czujnik wycofania tacki kropel
    lrLifterPullingPosition   : LREAL; //Pozycja podnośnika podczas przeciągania (podpinaj jeśli bDispencerWithLifter, innaczej pozostaw bez zmiennej)

    //WEJSCIA WYJSCIA SPRZETOWE
    // DO FML_READ
    // Struktura osi
    lrDropCatcherHeightCV : LREAL; 	// Aktualna wysokość tacki okapowej
    eDropCatcherState	 : E_Station; // Aktualny stan
	
	//StepMode
	bStepMode				: BOOL;		//Włączony tryb skokowy sterowania podnośnikami (tylko w serwisie)
	lrSetPosStepMode		: LREAL; 	//Ruch podnośnika o zadaną wartość w trybie krokowym (tylko w serwisie)

    //WEJSCIA WYJSCIA SPRZETOWE
    iStationIndex : UDINT;  //Numer stacji 
    sStationName  : WSTRING; //Nazwa stacji
	bSimDoser	:BOOL;
	
END_VAR
VAR_OUTPUT
    eState                 : E_Station;        //Stan ogólny bloku	
    eRunningState          : E_DispencerState; //Stan dozownika
    bError                 : BOOL;             //Błąd stacji
    nErrorNr               : UDINT;            //Nr błędu dozownika
    sErrorDescription      : STRING(200);      //Opis błędu
    sErrorDescription2     : STRING(200);      //Opis błędu
    sErrorStationName      : STRING;           //Nazwa stacji	
	udiStationID			: UDINT;				// Nr stacji
    nDispencerServoErrorNr : UDINT;            //Nr błędu serwo nalewarki
    nLifterServoErrorNr    : UDINT;            //Nr błędu serwo podnośnika
    lrDosedMassCV          : LREAL;            //Aktualna wydozowana doza
    bSuckingValveActuator  : BOOL;             //Siłownik zaworu ssącego
    bDosingValveActuator   : BOOL;             //Siłownik Zaworu tłoczącego
    bDropCatcherActuator   : BOOL;             //Siłownik tacki kropel	
    tCycleTime             : TIME;
    bCyclePrepareDone      : BOOL;
    bCycleDone             : BOOL;
    bCycleNotDone          : BOOL;
    bDosingDoneDelayOutput : BOOL;

    lrLifterActualPosition : LREAL; // Aktualna pozycja podnosnika dozownika
    bEncoderHomed          : BOOL;  // Dozowniki zbazowane
    bHomingDone            : BOOL;  //Wymagane ponowne bazowanie (blad podczas bazowania lub stop awaryjny)
    bMultiMasterSyncOut    : BOOL;  //OPCJA Synchronizacja gotości dozownika
END_VAR
VAR_IN_OUT

    //Fazy dozownika przy dozowaniu i ssaniu - jeśli wartości równe 0 faza zostanie pominięta. Następujące fazy muszą być od siebie większe	
    lrDosePhase1Volume        : LREAL; //Faza 1 dozowania (Podnośnik nieruchomy), do jakiej objętości ma trwać w [ml], następnie zaczyna sie 2 faza (powinna być mniejsza niż zadana objętość)
    lrDosePhase2Volume        : LREAL; //Faza 2 dozowania (Podnośnik zsynchronizowany z dozownikiem), do jakiej objętości ma trwać w [ml], następnie zaczyna sie 3 faza (powinna być mniejsza niż zadana objętość dozowania i większa od fazy 1)
    lrDosePhase1Velocity      : LREAL; //Prędkość dozowania Fazy 1 [ml/s]
    lrDosePhase2Velocity      : LREAL; //Prędkość dozowania Fazy 2 [ml/s] 
    lrDosePhase3Velocity      : LREAL; //Prędkość dozowania Fazy 3 [ml/s] 
    lrSuckVelocity            : LREAL; //Prędkość zasysania [ml/s] 
    lrDosePhase1Acceleration  : LREAL; //Przyspieszenie dozowania Fazy 1 [ml/s2]
    lrDosePhase2Acceleration  : LREAL; //Przyspieszenie dozowania Fazy 2 [ml/s2] 
    lrDosePhase3Acceleration  : LREAL; //Przyspieszenie dozowania Fazy 3 [ml/s2] 
    lrSuckAcceleration        : LREAL; //Przyspieszenie zasysania [ml/s2] 
    lrDosePhase1Deceleration  : LREAL; //Zwalnianie dozowania Fazy 1 [ml/s2]
    lrDosePhase2Deceleration  : LREAL; //Zwalnianie dozowania Fazy 2 [ml/s2] 
    lrDosePhase3Deceleration  : LREAL; //Zwalnianie dozowania Fazy 3 [ml/s2] 
    nDosingDoneDelayTime      : UDINT; //Czas odpóźnienia wykonania dozy [ms]
    lrSuckDeceleration        : LREAL; //Zwalnianie zasysania [ml/s2] 
    lrSuckValveOpenVolume     : LREAL; //Otwarcie zaworu ssącego po zadanej odległości od początku ssania [ml]
    lrSuckValveCloseVolume    : LREAL; //Zamknięcie zaworu ssącego po zadanej odległości od końca ssania [ml]
    lrDosingValveOpenVolume   : LREAL; //Otwarcie zaworu tłoczącego po zadanej odległości od początku tłoczenia [ml]
    lrDosingValveCloseVolume  : LREAL; //Zamknięcie zaworu tłoczącego po zadanej odległości od końca tłoczenia [ml]
	lrCatchHeightSV			  : LREAL; //Pozycja chwytaka
    lrLifterReadyPosition     : LREAL; //Pozycja podnośnika dozownika przy starcie dozowania (podpinaj jeśli bDispencerWithLifter, innaczej pozostaw bez zmiennej)
    lrLifterStartDosePosition : LREAL; //Pozycja podnośnika dozownika przy starcie dozowania (podpinaj jeśli bDispencerWithLifter, innaczej pozostaw bez zmiennej)
    lrLifterStopDosePosition  : LREAL; //Pozycja podnośnika dozownika przy starcie dozowania (podpinaj jeśli bDispencerWithLifter, innaczej pozostaw bez zmiennej)
    lrLifterVelocity          : LREAL; //Prędkość podnosnika dozownika (podpinaj jeśli bDispencerWithLifter, innaczej pozostaw bez zmiennej)
    lrLifterAcceleration      : LREAL; //Przyspieszenie podnośnika dozownika(podpinaj jeśli bDispencerWithLifter, innaczej pozostaw bez zmiennej)
    lrLifterDeceleration      : LREAL; //Zwalnianie podnośnika dozownika  (podpinaj jeśli bDispencerWithLifter, innaczej pozostaw bez zmiennej)
  

    lrSuckValveOpenTimeDelay  : LREAL := 0; (*NOWA 0-1000*) // [3] Opóżnienie rozpoczęcia ssania po tłoczeniu [ms]
    lrSuckValveCloseTimeDelay : LREAL := 0; (*NOWA 0-2000*) // [4] Opóżnienie zamknięcia zaworu ssącego [ms]
    lrDoseValveOpenTimeAcc    : LREAL := 0; (*NOWA 0-500*)  // [1] Przyśpieszenie otwarcia zaworu tłoczenia [ms]
    lrDoseValveCloseTimeDec   : LREAL := 0; (*NOWA 0-1000*) // [2] Opóźnienie zamknięcia zaworu tłoczenia [ms]
    lrDoseSuckingVolume       : LREAL := 0; (*NOWA 0-100*)  // [5] [Podsysanie] Wartość dozy do posysenia [ml]	
    lrDoseSuckingTimeDelay    : LREAL := 0; (*NOWA 0-500*)  // [6] [Podsysanie] Opóźnienie podsysania [ms]
    bDoseSucking              : BOOL; (*NOWA*)              // [Podsysanie] Opcja podsysania przy dozowaniu

    //Ruchy ręczne
    bManualMovement           : BOOL;  //Zezwolenie na ruchy ręczne
	bManualSync				  : BOOL;	// Synchronizacja-Przejazd tłoka i podnośnika do określonej pozycji
    lrManualOverride          : LREAL; //Procentowa redukcja prędkości wszystkich serw (Tylko w trybie serwisowym)
    bManualPullingFast        : BOOL;  //Przeciąganie dozownika szybkie
    bManualPullingSlow        : BOOL;  //Przeciąganie dozownika wolne
	bManualCleaningMode		  : BOOL;	//Włączenie trybu mycia
	bManualCleaning			  : BOOL;	//Włącz mycie, do synchronizacji
    bManualPistonBack         : BOOL;  //Ruch ręczny podnośnikiem stacji w górę
    bManualPistonForward      : BOOL;  //Ruch ręczny podnośnikiem stacji w dół
    bManualSuckingValve       : BOOL;  //Otwarcie ręczne zaworu ssącego
    bManualDosingValve        : BOOL;  //Otwarcie ręczne zaworu dozującego (iglicy)
    bManualDropCatcherForward : BOOL;  //Wysunięcie ręczne tacki kropel
    bManualLifterUp           : BOOL;  //Podniesienie ręczne stacji dozownika (podpinać zmienną jeśli bDispencerWithLifter=TRUE)
    bManualLifterDown         : BOOL;  //Opuszczenie ręczne stacji dozownika (podpinać zmienną jeśli bDispencerWithLifter=TRUE)

    //Struktury NC
    DispencerAxisRef       : AXIS_REF; //Struktura sterowania NC dla serwa Dozownika
    DispencerLifterAxisRef : AXIS_REF;
    //Hamulec
    bServiceBrakeOff : BOOL; //Wyłączenie serwisowe hamulca  

END_VAR
VAR
    mcDispencerMoveAbsolute1 : MC_MoveAbsolute; // Blok nr 1 ruchu absolutnego tłoka dozownika
    mcDispencerMoveAbsolute2 : MC_MoveAbsolute; // Blok nr 2 ruchu absolutnego tłoka dozownika
    mcDispencerManualMove    : MC_JOG;          // Blok ruchu manualnego tłokiem dozownika
    mcDispencerStop          : MC_Stop;         // Blok zatrzymania tłoka dozownika, jeśli to konieczne
    mcDispencerSoftReset     : MC_Reset;        // Blok łagodnego resetu serwa tloka dozownika
    mcDispencerPower         : Mc_Power;        // Blok zasilania serwa dozownika
    bDispencerServoPower     : BOOL;            // Zalaczenie zasilania serwa
    // Blok resetowania twardego błędu
    fbDispencerHardReset : FB_SoEReset;
    // Blok Resetowania twardego błędu podnośnika

    // Pozycja przy rozpoczeciu dozowania
    lrStartDosingPos : LREAL;
    // Pozycja startowa tłoka dozownika przy rozpoczęciu zasysania
    lrSuckingMassStart : LREAL;
    // Ruch absolutny fazy 3
    mcDispencerMoveAbsolute3 : MC_MoveAbsolute;
    tonCycleTimer            : TON;
    rtrigCycleTimerRead      : R_TRIG;
    // zablokowanie przeciągania
    bManualPullingLatch : BOOL;
    // Opóźnienie przejścia do stanu zakończenia dozowania
    tonDosingDoneDelay : TON;
    bStopped           : BOOL;

    tonSuckingValveCloseError : TON; // Błąd zamknięcia zaworu ssącego
    tonSuckingValveOpenError  : TON; // Błąd otwarcia zaworu ssącego
    tonDosingValveCloseError  : TON; // Błąd zamknięcia zaworu dozującego
    tonDosingValveOpenError   : TON; // Błąd otwarcia zaworu dozującego

    tonSuckValveOpenTimeDelay  : TON;
    tonSuckValveCloseTimeDelay : TON;
    tonDoseValveOpenTimeAcc    : TON;
    tonDoseValveCloseTimeDec   : TON;
    tonDoseSuckingTimeDelay    : TON;

    (**********FESTO PODNOŚNIK ******************)
    // Blok Resetowania twardego błędu podnośnika
    fbLifterHardReset : FB_SoEReset;
    // Blok miekkiego resetu serwa podnosnika
    mcLifterSoftReset : MC_Reset;
    // Blok ruchu absolutnego podnosnika
    mcLifterMoveAbsolute : MC_MoveAbsolute;
    mcLifterMoveAbsolute2 : MC_MoveAbsolute;	
    // Blok ruchu manualnego podnosnika
    mcLifterManualMove : MC_JOG;
    // Blok stopu podnosnika
    mcLifterStop : MC_Stop;
    // Blok zasilania serwa podnosnika
    mcLifterPower : Mc_Power;
    // Blok sprzęgania Dozownka z podnoszeniem
    mcLifterGearIn : Mc_GearInDyn;
    // Współczynnika przkeładni przy sprzeganiu dozownika z podnosnikiem (Wyliczany)
    lrGearRatio : LREAL;
    // Blok wysprzeglania dozownika i podnosnika
    mcLifterGearOut : Mc_GearOut;
    // Zasilanie serwo podnośnika dozownika
    bLifterServoPower     : BOOL;
    mcLifterGearInEnable  : BOOL;
    tofReset              : TOF;
	tonEstopDelay		  : TON;
    tonReadErrroFesto     : TON;
    rtLiftSynchroPh3      : R_TRIG;
    rtLiftSynchroPh2      : R_TRIG;
    rtLiftSynchroPh1      : R_TRIG;
    bPrepareToAborting    : BOOL;
    tonPrepareToAborting  : TON;
    lrPullingVelocity     : LREAL;
    TimerLifterNotEnabled : TON;
    rtDosingPh1           : R_TRIG;
    rtDosingPh2           : R_TRIG;
    rtDosingPh3           : R_TRIG;
    rtGoingUp             : R_TRIG;
    rtPreparingToDose     : R_TRIG;

    //Zabezpieczenie niektórych błędów aby pojawiały się tylko w cyklu
    bErrorOnlyIfCycleOn     : BOOL;
    tonDropCatcherOpenError : TON;
	tonDropCatcherCloseError: TON;	
    tonStartHoming          : TON;
    lrLifterMaxHeight       : LREAL;
    lrLifterMinHeight       : LREAL;
    nCountCheckDisp1        : INT;
    nCheckCount123          : INT;
    nCheckCount124          : INT;
    nCheckCount125          : INT;
    ninttest                : INT;
    tonTooLongDosing        : TON;
    nCheckCount1233         : INT;
    nCheckCount1234         : INT;
    nCheckCount1235         : INT;
    nCheckCount1263         : INT;
    nCheckCount1236         : INT;
    tonEror10LifterNotReady : TON;
	tonError2				: TON;
    nCountErr9              : INT;
    tonEror9LifterNotReady  : TON;
    bStateError             : BOOL;
    eLastState              : E_Station;        //Stan ogólny bloku
    eLastRunningState       : E_DispencerState; //Stan podbloku
    eLastStateTemp          : E_Station;        //Stan ogólny bloku
    eLastRunningStateTemp   : E_DispencerState; //Stan podbloku
    bPreparingToDisable     : BOOL;
    btestgoingup            : INT;
	iCaseGoingUp			: INT;
    bCountTestDoz1          : INT;
    bCountTestDoz2          : INT;

    bHeightSetNotDone : BOOL;

    mcHeightManualMove : INT;
    nCountTest12       : INT;
    bTest              : BOOL;
    trzeciafaza        : LREAL;
    drugafaza          : LREAL;
    calosc             : LREAL;
    tonDelayServoOn    : TON;
	tonDelayEnable: TON;
	
	//Bazowanie 
	bHardwareHoming			: BOOL;
	mcHardwareHomingPower	: MC_Power;
	fbHardwareHoming		: FB_HomingTorque;	

	//Step Mode
	rtStepModeUp			: R_TRIG;
	rtStepModeDown			: R_TRIG;
	lrStepModeHeightMotorSV	: LREAL;
	bStepModeMoving			: BOOL;
	tofStepModeMoving		: TOF;
	iManualSyncCase			: INT;
	bSucking 				: BOOL;
	
	//Podwójna doza
	bSecondDoseMode			: BOOL;
	iSecondDoseCount		: INT;
	bDoSecondDose			: BOOL;
	
	//Dodatkowe zasysanie
	bDoSmallSuckingOption	: BOOL;
	bDoSmallSucking			: BOOL;
	bDoSmallSuckingDone		: BOOL;	
	nDispencerError			: INT;
	nDispencerLifterError	: INT;
	bLifterIsNearReadyPosition: BOOL;
	
		//Zmienne od EVENTLOGGER
	bAlarmInit 						: BOOL := TRUE; 
	nAlarmNumerator					: INT;
	arfbAlarm						: ARRAY[0..19] OF  FB_TcAlarm;		//Tablica bloczków błędów
	fbSourceInfo 					: FB_TcSourceInfo;
	iSourceInfo						: I_TcSourceInfo;
	sAlarmTest						: STRING;
	//Koniec zmiennych od EVENTLOGGER
	tonbDispenserSim	:TON;
	tonbDispencerLifterSim	:ton;
END_VAR

IF NOT bHardwareHoming THEN
	Signals();
	SecondDose();
	ErrorHandling();
	Control();
	Limits();
	DispencerControlBlocks();
	IF bDispencerWithLifter THEN 
		LifterControlBlocks();	
	END_IF
ELSE
	HardwareHoming();
	DispencerAxisRef();
	DispencerAxisRef.NcToPlc.ActTorque;
	DispencerAxisRef.NcToPlc.ActPos;
	DispencerAxisRef.Status.Homed;
END_IF
AntyColision();
Statistics();
aStationID();


(*wypracowanie sygnałów wyjściowych z bloku*)
lrLifterActualPosition:=DispencerLifterAxisRef.NcToPlc.ActPos; 	//Pozycja 
//bHomingDone:=Lifter_FHPP_CTRL.HomingValid; DP

(*Przepisywanie aktualnie wydozowanej ilości do butelki*)
//1,2,3 faza
IF eRunningState>6 AND eRunningState<11 THEN
	lrDosedMassCV:=DispencerAxisRef.NcToPlc.ActPos-lrDoseVolume;
ELSE
	lrDosedMassCV:=0;
END_IF
(*Koniec przepisywanie aktualnie wydozowanej ilości do butelki*)

(*Zapisywanie ostatniego stanu*)
IF eLastStateTemp<>eState THEN
	eLastState := eLastStateTemp;
END_IF
eLastStateTemp := eState;
IF eLastRunningStateTemp<>eRunningState THEN
	eLastRunningState := eLastRunningStateTemp;
END_IF
eLastRunningStateTemp := eRunningState;
(*Koniec Zapisywanie ostatniego stanu*)

ACTION AntyColision:
(*Zabezpieczenie przed kolizją stacji poprzez ruch podnośnika*)	
IF bManualLifterDown AND DispencerLifterAxisRef.NcToPlc.ActPos<=lrMinPosition AND NOT bHoming AND NOT bHeightSet THEN
	bManualLifterDown:=FALSE;
END_IF	

IF bManualLifterUp AND DispencerLifterAxisRef.NcToPlc.ActPos>=lrMaxPosition AND NOT bHoming AND NOT bHeightSet THEN
	bManualLifterUp:=FALSE;
END_IF
END_ACTION

ACTION aStationID:
udiStationID	:=	iStationIndex;
END_ACTION

ACTION Control:
IF NOT bRUN THEN
				lrGearRatio:=-ABS(lrLifterStopDosePosition-lrLifterStartDosePosition+0.000000000001)
							/(*---------------------------------------------------------------------*)
							((BOOL_TO_INT(bLiftSynchroPh1)*lrDosePhase1Volume)
							+(BOOL_TO_INT(bLiftSynchroPh2)*(lrDoseVolume-lrDosePhase2Volume-lrDosePhase1Volume))
							+((BOOL_TO_INT(bLiftSynchroPh3)*(lrDoseVolume-lrDosePhase1Volume)))
							+ 0.000000000001); 					
	drugafaza:=(lrDoseVolume-lrDosePhase2Volume-lrDosePhase1Volume);						
	trzeciafaza:=(lrDoseVolume-lrDosePhase2Volume);
	calosc:=(*---------------------------------------------------------------------*)
							((BOOL_TO_INT(bLiftSynchroPh1)*lrDosePhase1Volume)
							+(BOOL_TO_INT(bLiftSynchroPh2)*(lrDoseVolume-lrDosePhase2Volume-lrDosePhase1Volume))
							+((BOOL_TO_INT(bLiftSynchroPh3)*lrDosePhase2Volume))
							+ 0.000000000001);
END_IF
	



	(** TIMERY**)
	tonDoseValveOpenTimeAcc(	IN:= eRunningState = E_DispencerState.eDosingPh1, 											PT:= LREAL_TO_TIME(lrDoseValveOpenTimeAcc));   		// [1] Przyśpieszenie otwarcia zaworu tłoczenia [ms]
	tonDoseValveCloseTimeDec(	IN:= (eRunningState=E_DispencerState.eDosingPh3 AND NOT bDoseSucking) OR
									 (eRunningState=E_DispencerState.eDoseSucking AND mcDispencerMoveAbsolute1.Done),		PT:= LREAL_TO_TIME(lrDoseValveCloseTimeDec));  		// [2] Opóźnienie zamknięcia zaworu tłoczenia [ms]
	tonSuckValveOpenTimeDelay(	IN:= eRunningState = E_DispencerState.eGoingUp,											PT:= LREAL_TO_TIME(lrSuckValveOpenTimeDelay));		// [3] Opóżnienie rozpoczęcia ssania po tłoczeniu [ms]
	tonSuckValveCloseTimeDelay(	IN:= (bSucking) AND
//										 (mcDispencerMoveAbsolute1.Done OR NOT mcDispencerMoveAbsolute1.Execute), 		PT:= LREAL_TO_TIME(lrSuckValveCloseTimeDelay)); 	// [4] Opóżnienie zamknięcia zaworu ssącego [ms]
										 (mcDispencerMoveAbsolute1.Done OR NOT mcDispencerMoveAbsolute1.Busy), 			PT:= LREAL_TO_TIME(lrSuckValveCloseTimeDelay)); 	// [4] Opóżnienie zamknięcia zaworu ssącego [ms]
	tonDoseSuckingTimeDelay(	IN:= eRunningState = E_DispencerState.eDoseSucking,										PT:= LREAL_TO_TIME(lrDoseSuckingTimeDelay));    	// [6] [Podsysanie] Opóźnienie podsysania [ms]

	//Opóźnienie potwierdzenia wykonania dozy
	(*tonDosingDoneDelay(IN:=(eRunningState=E_DispencerState.eDosingDone OR eRunningState=E_DispencerState.eSucking)AND
							mcDispencerMoveAbsolute1.Done AND tonSuckValveCloseTimeDelay.Q 				
							, PT:=UDINT_TO_TIME(nDosingDoneDelayTime));*)
	tonPrepareToAborting(IN:=bPrepareToAborting, PT:=T#1S);
	//Opóźnienie potwierdzenia wykonania dozy Zmiana 20200820
//	tonDosingDoneDelay(IN:=(eRunningState=E_DispencerState.eDosingDone OR eRunningState=E_DispencerState.eSucking)				
//							, PT:=UDINT_TO_TIME(nDosingDoneDelayTime));
	tonDosingDoneDelay(IN:=(eRunningState=E_DispencerState.eGoingUp AND iCaseGoingUp = 30)				
							, PT:=UDINT_TO_TIME(nDosingDoneDelayTime));
	
							
	tonDelayServoOn(IN:=(eState = E_Station.ePreparingToReady), PT:=T#7S); //Nowe XTS bylo 1200ms						
	tonDelayEnable(IN:=	bEnable, PT:=T#5S);			
	(*Synchronizacja tylko jedna zaznaczona*)
	(*Zabezpieczenie przed zalaczeniem trzech*)
(*	rtLiftSynchroPh3(CLK:=bLiftSynchroPh3,Q=>);rtLiftSynchroPh2(CLK:=bLiftSynchroPh2,Q=>);rtLiftSynchroPh1(CLK:=bLiftSynchroPh1,Q=>);
	IF rtLiftSynchroPh1.Q THEN	bLiftSynchroPh2:=FALSE;	bLiftSynchroPh3:=FALSE; END_IF
	IF rtLiftSynchroPh2.Q THEN	bLiftSynchroPh1:=FALSE;	bLiftSynchroPh3:=FALSE; END_IF
	IF rtLiftSynchroPh3.Q THEN	bLiftSynchroPh1:=FALSE;	bLiftSynchroPh2:=FALSE; END_IF 
	IF bLiftSynchroPh1 THEN	bLiftSynchroPh2:=FALSE;	bLiftSynchroPh3:=FALSE;
	ELSIF bLiftSynchroPh2 THEN	bLiftSynchroPh1:=FALSE;	bLiftSynchroPh3:=FALSE;
	ELSIF bLiftSynchroPh3 THEN	bLiftSynchroPh1:=FALSE;	bLiftSynchroPh2:=FALSE;
	ELSIF NOT bLiftSynchroPh1  AND NOT bLiftSynchroPh2 AND NOT bLiftSynchroPh3 THEN	bLiftSynchroPh1:=TRUE;	bLiftSynchroPh2:=FALSE;	bLiftSynchroPh3:=FALSE; END_IF
	(*Koniec Zabezpieczenie przed zalaczeniem trzech*)
*)
	
	//	100					300			250
	IF lrDosePhase1Volume>lrDoseVolume-lrDosePhase2Volume THEN
		lrDosePhase1Volume:=lrDoseVolume-lrDosePhase2Volume;
	END_IF
	// 200					300			200
	IF lrDosePhase2Volume>lrDoseVolume-lrDosePhase1Volume THEN
		lrDosePhase2Volume:=lrDoseVolume-lrDosePhase1Volume;
	END_IF
	
	IF  eState=E_Station.eReady OR eRunningState=E_DispencerState.eDosingDone OR eRunningState=E_DispencerState.eGoingUp THEN
//	IF  (eState>E_Station.eError AND eState<=E_Station.eReady) OR eRunningState=E_DispencerState.eDosingDone OR eRunningState=E_DispencerState.eGoingUp THEN
		IF (DispencerLifterAxisRef.NcToPlc.ActPos  >= lrDropCatcherHeightCV+(lrDropCatcherOpenDistance-5)) AND lrDropCatcherHeightCV>1 AND NOT bHoming AND NOT bHeightSet THEN
			bDropCatcherActuator:=TRUE;
		ELSE
			bDropCatcherActuator:=FALSE;
		END_IF
	END_IF
							
							
	//Zbocza 
	rtDosingPh1(CLK:=eRunningState=E_DispencerState.eDosingPh1,Q=>);
	rtDosingPh2(CLK:=eRunningState=E_DispencerState.eDosingPh2,Q=>);
	rtDosingPh3(CLK:=eRunningState=E_DispencerState.eDosingPh3,Q=>);
	rtGoingUp(CLK:=eRunningState=E_DispencerState.eGoingUp,Q=>);
	rtPreparingToDose(CLK:=eRunningState=E_DispencerState.ePreparingToDose,Q=>);	
	
	(*****Wyłączenie enable*****)
	IF NOT bEnable THEN
		IF eState <> E_Station.eDisabled AND eState <> E_Station.ePreparingToDisable THEN
			eState 				:= E_Station.ePreparingToDisable; 
			bCycleDone			:= FALSE;
		END_IF	
	END_IF

	(*****Estop*****)
	IF (NOT bEstop AND bInLimitSwitchSensor) OR (NOT bEStopButtonsAndDoors AND NOT bInLimitSwitchSensor) THEN	
		IF eState <> E_Station.eAborted AND eState <> E_Station.eAborting AND eState <> E_Station.eDisabled THEN
			eState 				:= E_Station.eAborting; 
		END_IF
	END_IF

	
	CASE eState OF
	/////////////////////////////	
		E_Station.eDisabled: 					// Stan nieaktywnosci (Stacja wyłączona) 
		
			IF bEnable AND tonDelayEnable.Q THEN
				eState 				:= E_Station.ePreparingToReady; 
			END_IF 
			
    /////////////////////////////	    
		E_Station.eAborted: 					// Stan bezpiecznego zatrzymania (po Abortingu) 

			IF bEStop THEN
				eState 				:= E_Station.ePreparingToReady;
			END_IF
			
	/////////////////////////////	
		E_Station.eAborting:                 	// Stan bezpiecznego zatrzymywania (po EStopie)
		
			mcDispencerPower.Override			:= 100;
			mcDispencerStop.Execute				:= NOT bStopped AND bDispencerServoPower; //Nowe XTS
			mcDispencerMoveAbsolute1.Execute	:= FALSE;
			mcDispencerMoveAbsolute2.Execute	:= FALSE;
			mcDispencerManualMove.JogBackwards	:= FALSE;
			mcDispencerManualMove.JogForward	:= FALSE;			
			
			IF bDispencerWithLifter THEN (*n*)
				mcLifterPower.Override				:= 100;
				mcLifterStop.Execute				:= NOT bStopped AND bLifterServoPower; //Nowe XTS
				mcLifterMoveAbsolute.Execute		:= FALSE;	
				mcLifterManualMove.JogBackwards		:= FALSE;
				mcLifterManualMove.JogForward		:= FALSE;
				bHeightSetNotDone 					:= FALSE; //Zmiana 2021-02-19
			END_IF	
											(*n*)					//Zmiana XTS
			IF ((mcLifterStop.Done OR NOT bDispencerWithLifter OR NOT bLifterServoPower) AND (mcDispencerStop.Done OR NOT bDispencerServoPower)) OR bStopped THEN
				
				mcDispencerStop.Execute			:=	FALSE;
				bDispencerServoPower			:=	FALSE;
				
				mcLifterStop.Execute			:=	FALSE;
				bLifterServoPower				:=	FALSE;
				
				bStopped						:=	FALSE;
				eState							:=	E_Station.eAborted; 
				eRunningState					:=	E_DispencerState.eReady;
			END_IF	
					
	/////////////////////////////			
		E_Station.eError:                 	 	// Stan błędu 	
			
			IF bReset OR tofReset.Q THEN
				eState 				:= E_Station.eResetting;
				eRunningState		:= E_DispencerState.eReady;
			ELSE
				ResetCommands();
				mcLifterSoftReset	(Execute:=FALSE,Axis:=DispencerLifterAxisRef);
				mcDispencerSoftReset(Execute:=FALSE,Axis:=DispencerAxisRef);
			END_IF
			
	/////////////////////////////
		E_Station.eResetting:					// Stan resetowania bledu (po Errorze)
			
			//Procedura obsługi resetu w zależności od błędu
// 			CASE nErrorNr OF
// //			CASE nErrorNr-iStationIndex OF
// 		
// 				//Error 2 - BŁĄD SERWA DOZOWNIKA
// 				141:
// 				Alarm_0220	220	Error	Błąd napędu tłoka - upewnij się że został dobrze złożony. Błąd NC: {0}	
				IF arfbAlarm[0].bActive THEN	
					mcDispencerSoftReset(Execute:=TRUE,Axis:=DispencerAxisRef);
					IF mcLifterGearIn.InGear THEN
						mcLifterGearIn.Enable:=FALSE;
						mcLifterGearOut.Execute := TRUE;
					END_IF
					IF mcLifterGearOut.Done THEN
						mcLifterGearOut.Execute := FALSE;
					END_IF
					IF NOT mcLifterGearIn.InGear AND NOT mcLifterGearOut.Execute THEN
					
						IF NOT fbDispencerHardReset.Busy AND NOT mcDispencerSoftReset.Busy AND mcDispencerPower.Status AND NOT DispencerAxisRef.Status.Error THEN
								mcDispencerSoftReset(Execute:=FALSE,Axis:=DispencerAxisRef);
								nErrorNr:=0;
								nDispencerServoErrorNr:=0;
								bError := FALSE;
								sErrorDescription:='';	
				
						ELSIF NOT fbDispencerHardReset.Busy AND NOT mcDispencerSoftReset.Busy AND NOT mcDispencerPower.Status AND NOT DispencerAxisRef.Status.Error THEN
								nErrorNr:=0;
								nDispencerServoErrorNr:=0;
								bError := FALSE;
								sErrorDescription:='';
						END_IF
						IF fbDispencerHardReset.Error OR mcDispencerSoftReset.Error THEN
							mcDispencerSoftReset(Execute:=FALSE,Axis:=DispencerAxisRef);
						END_IF
						
					END_IF
				END_IF
				// Alarm_0221	221	Error	Błąd napędu podnośnika. Błąd NC: {0}
				//Error 2, Error 4 - BŁĄD SERWA PODNOSZENIA DOZOWNIKA
//				142:	
				IF arfbAlarm[1].bActive THEN
					mcLifterGearIn.Enable:=FALSE;
					mcLifterGearOut.Execute:=FALSE;
					//fbLifterHardReset(Execute:=NOT mcLifterMoveAbsolute.Execute,Axis:=DispencerLifterAxisRef);
					mcLifterSoftReset(Execute:=NOT mcLifterMoveAbsolute.Execute,Axis:=DispencerLifterAxisRef);
					IF NOT fbLifterHardReset.Busy AND NOT mcLifterSoftReset.Busy AND mcLifterPower.Status AND NOT DispencerLifterAxisRef.Status.Error THEN
						//fbLifterHardReset(Execute:=FALSE,Axis:=DispencerLifterAxisRef);
						mcLifterSoftReset(Execute:=FALSE,Axis:=DispencerLifterAxisRef);
						bDropCatcherActuator 					:= FALSE;
						IF bDropCatcherBackSensor THEN
							mcLifterMoveAbsolute.Execute		:= TRUE;
						END_IF
						mcLifterMoveAbsolute.Acceleration	:=	lrLifterAcceleration/15;
						mcLifterMoveAbsolute.Velocity		:=	lrLifterVelocity/15;						
						mcLifterMoveAbsolute.Position		:=	lrLifterReadyPosition;
						mcLifterPower.Override:=100; 
						IF mcLifterMoveAbsolute.Done THEN
							bDropCatcherActuator:=TRUE;
							mcLifterPower.Override:=100; 
							mcLifterMoveAbsolute.Execute:=FALSE;
							nErrorNr:=0;
							nLifterServoErrorNr:=0;
							bError := FALSE;
							sErrorDescription:='';	
						END_IF 
					ELSIF NOT fbLifterHardReset.Busy AND NOT mcLifterSoftReset.Busy AND NOT mcLifterPower.Status AND NOT DispencerLifterAxisRef.Status.Error THEN		
						//fbLifterHardReset(Execute:=FALSE,Axis:=DispencerLifterAxisRef);
						mcLifterSoftReset(Execute:=FALSE,Axis:=DispencerLifterAxisRef);
						nErrorNr:=0;
						nLifterServoErrorNr:=0;
						bError := FALSE;
						sErrorDescription:='';	
					END_IF
					IF fbLifterHardReset.Error OR mcLifterSoftReset.Error THEN
						//fbLifterHardReset(Execute:=FALSE,Axis:=DispencerLifterAxisRef);
						mcLifterSoftReset(Execute:=FALSE,Axis:=DispencerLifterAxisRef);
					END_IF	
				END_IF
				// inny numer błędu
				IF NOT arfbAlarm[0].bActive AND NOT arfbAlarm[1].bActive THEN
					bSuckingValveActuator:=FALSE;
					bDosingValveActuator:=FALSE;
					IF bDispencerWithLifter THEN
						mcLifterSoftReset(Execute:=FALSE,Axis:=DispencerLifterAxisRef);
						mcLifterPower.Override				:=	100; 
						mcLifterMoveAbsolute.Acceleration	:=	lrLifterAcceleration/15;
						mcLifterMoveAbsolute.Velocity		:=	lrLifterVelocity/15;
						mcLifterMoveAbsolute.Position		:=	lrLifterReadyPosition;
						bDropCatcherActuator				:=	FALSE;
						IF bDropCatcherBackSensor THEN
							mcLifterMoveAbsolute.Execute:=	bLifterServoPower;
						END_IF						
						
						IF mcLifterMoveAbsolute.Done OR NOT bLifterServoPower THEN 
							bDropCatcherActuator:=TRUE;
							mcLifterPower.Override:=100; 
							mcLifterMoveAbsolute.Execute:=FALSE;
							nErrorNr:=0;
							nLifterServoErrorNr:=0;
							bError := FALSE;
							sErrorDescription:='';	
						END_IF
					ELSE
						bError := FALSE;
					END_IF 
			END_IF
// 			END_CASE	
			
			IF NOT bError THEN
				nErrorNr 			:=	0;
   				sErrorDescription 	:=	'';
	
				eState 				:=	E_Station.ePreparingToReady;
			ELSE
				eState 				:=	E_Station.eError;
			END_IF
        
	/////////////////////////////
		E_Station.eManualMovement:     			// Stan ruchów manualnych  
       
			ManualMovements();
			//Wyjście z trybu serwisowego
			IF NOT bManualMovement AND bInLimitSwitchSensor  AND NOT bChangeover THEN
				mcDispencerPower.Override			:=	100;		
				bSuckingValveActuator				:=	FALSE;
				bDosingValveActuator				:=	FALSE;
				mcDispencerMoveAbsolute1.Execute	:=	FALSE;
			
				IF bDispencerWithLifter THEN
					IF lrLifterActualPosition < lrLifterReadyPosition - 1 THEN
						bDropCatcherActuator				:=	FALSE;
						IF bDropCatcherBackSensor THEN
							mcLifterMoveAbsolute.Execute	:=	 TRUE;
						END_IF						
						mcLifterMoveAbsolute.Acceleration	:= lrLifterAcceleration/15;
						mcLifterMoveAbsolute.Velocity		:= lrLifterVelocity/15;
						mcLifterMoveAbsolute.Position		:= lrLifterReadyPosition;
					END_IF
				END_IF
				
				IF NOT bDispencerWithLifter OR mcLifterMoveAbsolute.Done OR lrLifterActualPosition >= lrLifterReadyPosition THEN
					mcDispencerMoveAbsolute1.Execute:=FALSE;
					mcLifterMoveAbsolute.Execute	:=FALSE;
					eState 							:= E_Station.eReady;
					iManualSyncCase					:= 0;
					eRunningState					:=	E_DispencerState.eReady;
				END_IF
			END_IF

	/////////////////////////////
		E_Station.eHoming:						// Stan bazowania 

			Homing();
			IF NOT bHoming AND NOT bHeightSet THEN
			   eState:=E_Station.ePreparingToReady;
			   	mcLifterManualMove.JogForward		:= FALSE;
				mcLifterManualMove.JogBackwards		:= FALSE;
			END_IF			
			
	/////////////////////////////
		E_Station.eHomingDone:                  // Stan wykonania bazowania 
		
			bHomingDone							:=	TRUE;
			IF NOT bHoming AND NOT bHeightSet THEN
				
			   eState:=E_Station.eReady;
			END_IF
			
	/////////////////////////////
		E_Station.ePreparingToReady:            // Stan przygotowywania do gotowosci (zawsze przed Ready)  

		
			IF tonDelayServoOn.Q THEN
				bDispencerServoPower		:= TRUE;		
				bLifterServoPower			:= TRUE;//bDispencerWithLifter	; (*n*) //ZMIANA XTS
			END_IF	
		
			mcDispencerPower.Override	:= 100;
			bDosingValveActuator		:= FALSE;
			bSuckingValveActuator		:= FALSE;
			bManualDosingValve			:= FALSE;
			bManualSuckingValve			:= FALSE;
			bServiceBrakeOff			:= FALSE;

			mcLifterMoveAbsolute.Execute := FALSE;

			mcDispencerMoveAbsolute1.Execute := FALSE;
			mcDispencerMoveAbsolute2.Execute := FALSE;
			mcDispencerMoveAbsolute3.Execute := FALSE;
				(*n*)
			IF (mcLifterPower.Status OR NOT bDispencerWithLifter) AND mcDispencerPower.Status THEN
											(*n*)
				IF NOT bHeightSetNotDone AND bDispencerWithLifter THEN
					
					IF mcLifterGearIn.InGear THEN
						mcLifterGearIn.Enable := FALSE;
						mcLifterGearOut.Execute := TRUE;
					ELSIF mcLifterGearIn.Enable AND mcLifterGearOut.Done THEN 
						mcLifterGearOut.Execute := FALSE;
					ELSE

						mcLifterPower.Override:=100;
						mcLifterMoveAbsolute.Acceleration	:=	lrLifterAcceleration/15;
						mcLifterMoveAbsolute.Velocity		:=	lrLifterVelocity/15;
						
						bDropCatcherActuator			:=	FALSE;
						IF bDropCatcherBackSensor THEN
							mcLifterMoveAbsolute.Execute:=	TRUE;
						END_IF
						mcLifterMoveAbsolute.Position	:=	lrLifterReadyPosition;
						IF bChangeover THEN
							mcLifterMoveAbsolute.Position:=lrMaxPosition;
						END_IF
						IF mcLifterMoveAbsolute.Done THEN
							mcLifterMoveAbsolute.Execute:=FALSE;
							eState:=E_Station.eReady;
							eRunningState:=E_DispencerState.eReady;
						END_IF
					END_IF
					
				ELSE
					bHeightSetNotDone := FALSE;
					eState:=E_Station.eReady;
					eRunningState:=E_DispencerState.eReady;
				END_IF	
			END_IF
         	IF bIgnoreError THEN
				eState:=E_Station.eReady;
				eRunningState:=E_DispencerState.eReady;
			END_IF


	
				
	/////////////////////////////
		E_Station.ePreparingToDisable:          // Stan przygotowywania do nieaktywnosci (po wyłączeniu Enable) 
  			bDropCatcherActuator:=FALSE; //Zmiana 29072019
			mcDispencerPower.Override:=100;
			mcLifterPower.Override:=100;
			IF bPreparingToDisable THEN
				mcLifterStop.Execute:=FALSE;
				mcLifterMoveAbsolute.Execute:= NOT mcLifterStop.Execute AND NOT  mcLifterStop.DONE;
				mcLifterMoveAbsolute.Position:=lrMaxPosition;
				mcLifterMoveAbsolute.Acceleration:=lrLifterAcceleration/15;
				mcLifterMoveAbsolute.Deceleration:=lrLifterDeceleration;
				mcLifterMoveAbsolute.Velocity:=lrLifterVelocity/15;
				IF mcLifterMoveAbsolute.Done THEN
					mcLifterMoveAbsolute.Execute:=FALSE;
					eState:=E_Station.eDisabled;
					bPreparingToDisable := FALSE;
					bDispencerServoPower:=FALSE;
					bLifterServoPower:=FALSE;
				END_IF
			ELSE
				mcDispencerStop.Execute:=NOT mcDispencerMoveAbsolute1.Execute AND NOT mcDispencerMoveAbsolute2.Execute AND NOT mcDispencerMoveAbsolute3.Execute;
				mcDispencerMoveAbsolute1.Execute:=FALSE;
				mcDispencerMoveAbsolute2.Execute:=FALSE;
				mcDispencerMoveAbsolute3.Execute:=FALSE;
		
				IF 	mcDispencerStop.Done  THEN
								
					IF bDispencerWithLifter AND DispencerLifterAxisRef.NcToPlc.CoupleState<3 THEN
						mcLifterGearOut.Execute:=FALSE;
						mcLifterGearIn.Enable:=FALSE;			
						mcLifterStop.Execute:=NOT mcLifterMoveAbsolute.Execute;
						mcLifterMoveAbsolute.Execute:=FALSE;
						mcLifterStop.Execute:=TRUE;
					ELSIF  bDispencerWithLifter AND DispencerLifterAxisRef.NcToPlc.CoupleState=3 THEN
						mcLifterGearIn.Enable:=FALSE;
						mcLifterGearOut.Execute:=TRUE;
					END_IF
		
					IF bEstop AND (bDispencerWithLifter AND DispencerLifterAxisRef.NcToPlc.CoupleState<3) THEN
						bPreparingToDisable:=TRUE;
						bSuckingValveActuator:=FALSE;
						bDosingValveActuator:=FALSE;;
					
					ELSIF (NOT bDispencerWithLifter OR mcLifterStop.Done) AND mcDispencerStop.Done THEN
						bDispencerServoPower:=FALSE;
						bDropCatcherActuator:=FALSE;
						IF bDispencerWithLifter THEN
							bLifterServoPower:=FALSE;
							mcLifterGearOut.Execute:=FALSE;
							mcLifterStop.Execute:=FALSE;
						END_IF
						mcDispencerStop.Execute:=FALSE;
						eState:=E_Station.eDisabled;
						mcDispencerStop.Execute:=FALSE;
						
						bSuckingValveActuator:=FALSE;
						bDosingValveActuator:=FALSE;
					END_IF
				END_IF
			END_IF
			
	/////////////////////////////
		E_Station.eReady:						// Stan gotowosci 
			
			IF NOT bSucking AND bDoSmallSucking THEN
				mcDispencerMoveAbsolute1.Execute:= bDosingValveClosedSensor; 
				mcDispencerMoveAbsolute1.Velocity:= lrSuckVelocity;
				mcDispencerMoveAbsolute1.Position:= lrDoseVolume + 3;
				mcDispencerMoveAbsolute1.Acceleration:= lrSuckAcceleration;
				mcDispencerMoveAbsolute1.Deceleration:= lrSuckDeceleration;
				IF mcDispencerMoveAbsolute1.Done THEN
					bDoSmallSucking						:=	FALSE;
					bDoSmallSuckingDone					:=	TRUE;
					mcDispencerMoveAbsolute1.Execute	:=	FALSE;
				END_IF
			END_IF
		
			// ZASYWANIE PRZY ZJEZDZIE W DÓŁ
			IF  tonSuckValveCloseTimeDelay.Q  THEN  // [4] Opóżnienie zamknięcia zaworu ssącego [ms]                            
				bSucking := FALSE;
				mcDispencerMoveAbsolute1.Execute:= FALSE;
				bSuckingValveActuator:=FALSE;
			END_IF	
			
			IF NOT bDoSmallSucking THEN
				IF bRun AND NOT bCycleDone AND NOT bCycleNotDone THEN
					eState 				:= E_Station.eStarting; 
				END_IF
				IF bHoming OR bHeightSet THEN
					eState 				:= E_Station.eHoming; 
				END_IF
				IF bManualMovement OR NOT bInLimitSwitchSensor OR bChangeover THEN //Przejscie do serwisu jak nie ma na czujniku
					IF NOT bInLimitSwitchSensor THEN
						bLifterServoPower		:=	FALSE;
					END_IF
					//Jeśli przejście w tryb ruchów manualnych przepisz wszystkie stany siłowników sterowanych przez moduł
					//aby zapobiec ewentualnym kolizjom po wejściu w tryb serwisowy
					bManualDosingValve			:=	bDosingValveActuator;
					bManualSuckingValve			:=	bSuckingValveActuator;
					bManualDropCatcherForward	:=	bDropCatcherActuator;
					mcDispencerStop.Execute		:=	FALSE;
					//eState 						:=	E_Station.eManualMovement; 
				
					// Dodanie zmieny narzędzia, zamiast wyłączenia stacja jedzie do góry i będzie możliwość
					// tych samych funkcji co w trybie serwisowy, przeciągania itp
					IF bChangeover THEN
						IF bDispencerWithLifter THEN
								IF lrLifterActualPosition < lrMaxPosition + 1 THEN
								bDropCatcherActuator			:=	FALSE;
								IF bDropCatcherBackSensor THEN
									mcLifterMoveAbsolute.Execute:=	TRUE;
								END_IF
								mcLifterMoveAbsolute.Acceleration	:= lrLifterAcceleration/15;
								mcLifterMoveAbsolute.Velocity		:= lrLifterVelocity/15;
								mcLifterMoveAbsolute.Position		:= lrMaxPosition;
							END_IF
						END_IF
						
						IF NOT bDispencerWithLifter OR mcLifterMoveAbsolute.Done OR lrLifterActualPosition >= lrMaxPosition  THEN
							mcDispencerMoveAbsolute1.Execute	:=FALSE;
							mcLifterMoveAbsolute.Execute		:=FALSE;
							eState 						:=	E_Station.eManualMovement; 
						END_IF
					ELSE
						eState 						:=	E_Station.eManualMovement; 
					END_IF	
				
				END_IF
				IF NOT bRun THEN
					bCycleDone 					:= FALSE;
					bCycleNotDone 				:= FALSE;	
				END_IF
				
				bStopped						:= FALSE;
				mcLifterStop.Execute			:= FALSE;
				mcDispencerStop.Execute			:= FALSE;
				iSecondDoseCount				:= 0;
			END_IF
	/////////////////////////////
		E_Station.eStopping:					// Stan zatrzymywania 
			eRunningState:=E_DispencerState.eReady;//zmiana 20200820
			Running();
			
			mcDispencerPower.Override:=100;
			mcLifterPower.Override:=100;
			mcDispencerStop.Execute:= NOT mcDispencerMoveAbsolute1.Execute AND NOT mcDispencerMoveAbsolute2.Execute AND NOT mcDispencerMoveAbsolute3.Execute AND NOT mcDispencerStop.CommandAborted;
			mcDispencerMoveAbsolute1.Execute:=FALSE;
			mcDispencerMoveAbsolute2.Execute:=FALSE;
			mcDispencerMoveAbsolute3.Execute:=FALSE;
			IF mcDispencerStop.Done THEN
				bDosingValveActuator:=FALSE;
				bSuckingValveActuator:=FALSE;
				IF bDispencerWithLifter THEN
					mcLifterMoveAbsolute.Execute:=FALSE;
					mcLifterMoveAbsolute.BufferMode:=MC_Aborting;
					mcLifterGearIn.Enable:=FALSE;
					mcLifterGearOut.Execute:=TRUE;
					IF mcLifterGearOut.Done THEN; 				
						bDropCatcherActuator			:=	FALSE;
						IF bDropCatcherBackSensor THEN
							mcLifterMoveAbsolute.Execute:=	bStopped;
						END_IF										
						IF mcLifterStop.DONE THEN
							bStopped:=TRUE;
						END_IF
						mcLifterStop.Execute:=NOT bStopped;
						
						mcLifterMoveAbsolute.Acceleration:=lrLifterAcceleration/15;
						mcLifterMoveAbsolute.Velocity:=lrLifterVelocity/15;
						mcLifterMoveAbsolute.Position:=lrLifterReadyPosition;
						
						IF mcLifterMoveAbsolute.Done AND bStopped THEN
							//mcLifterMoveAbsolute.Execute:=FALSE;
							//mcLifterMoveAbsolute.BufferMode:=MC_Aborting;
							eState:=E_Station.eReady;
							bStopped:=FALSE;
							bDropCatcherActuator:=TRUE;
							mcDispencerStop.Execute:=FALSE;
							mcLifterMoveAbsolute.Execute:=FALSE;
							mcLifterGearOut.Execute:=FALSE;
						END_IF
					END_IF
				ELSE
					mcDispencerStop.Execute:=FALSE;
					eState:=E_Station.eReady;
				END_IF
			END_IF
	
			IF mcLifterMoveAbsolute.Error THEN
				mcLifterMoveAbsolute.Execute:=FALSE;
			END_IF
			
	/////////////////////////////
		E_Station.eStarting:                  	// Stan uruchamiania (po Ready)
		
			eState					 := E_Station.eRunning; 
			
	/////////////////////////////
		E_Station.eRunning:               		// Stan wykonywania cyklu (po Startingu), w tym stanie osobny
 
			Running();
			IF NOT bRun THEN					(*Przerywanie cyklu*)
				eState 				 := E_Station.eStopping;	
				bCountTestDoz1:=bCountTestDoz1+1;
			END_IF
			IF bCycleDone OR bCycleNotDone THEN (*Cykl zakończony*)
				eState 				 := E_Station.eReady;
				eRunningState		 := E_DispencerState.eReady;//zmiana 20200820
				bCountTestDoz2:=bCountTestDoz2+1;
			END_IF	
			
			
	/////////////////////////////		
	END_CASE
END_ACTION

ACTION DispencerControlBlocks:
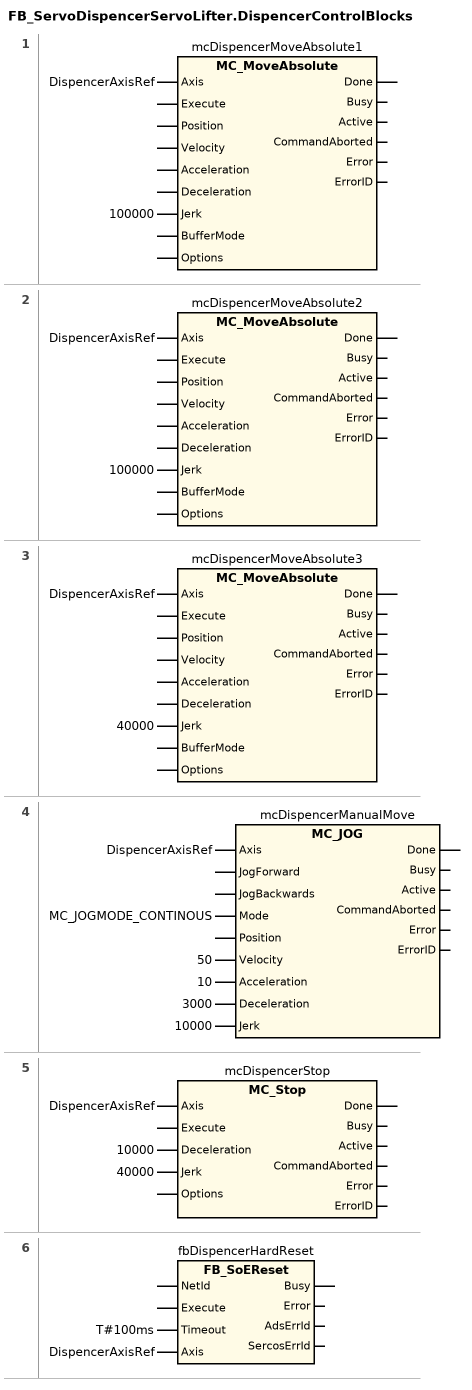
// NETWORK 1
mcDispencerMoveAbsolute1(Axis := DispencerAxisRef, Jerk := 100000); // MC_MoveAbsolute

// NETWORK 2
mcDispencerMoveAbsolute2(Axis := DispencerAxisRef, Jerk := 100000); // MC_MoveAbsolute

// NETWORK 3
mcDispencerMoveAbsolute3(Axis := DispencerAxisRef, Jerk := 40000); // MC_MoveAbsolute

// NETWORK 4
mcDispencerManualMove(
    Axis := DispencerAxisRef,
    Mode := MC_JOGMODE_CONTINOUS,
    Velocity := 50,
    Acceleration := 10,
    Deceleration := 3000,
    Jerk := 10000); // MC_JOG

// NETWORK 5
mcDispencerStop(Axis := DispencerAxisRef, Deceleration := 10000, Jerk := 40000); // MC_Stop

// NETWORK 6
fbDispencerHardReset(Timeout := T#100ms, Axis := DispencerAxisRef); // FB_SoEReset

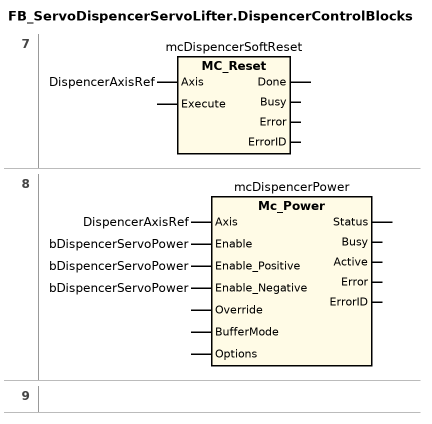
// NETWORK 7
mcDispencerSoftReset(Axis := DispencerAxisRef); // MC_Reset

// NETWORK 8
mcDispencerPower(
    Axis := DispencerAxisRef,
    Enable := bDispencerServoPower,
    Enable_Positive := bDispencerServoPower,
    Enable_Negative := bDispencerServoPower); // Mc_Power

// NETWORK 9
END_ACTION

ACTION ErrorHandling:
// Alarm_0220	220	Error	Błąd napędu tłoka - upewnij się że został dobrze złożony. Błąd NC: {0}		
// Alarm_0221	221	Error	Błąd napędu podnośnika. Błąd NC: {0}		
// Alarm_0222	222	Error	Nastawa dozy powyżej maksymalnej wartości - zmniejsz ilość dozy		
// Alarm_0223	223	Error	Nastawa dozy poniżej minimalnej wartość - zwiększ ilość dozy		
// Alarm_0224	224	Error	Zacięcie zaworu zasysania podczas zamykania - sprawdź czujnik		
// Alarm_0225	225	Error	Zacięcie zaworu zasysania masy podczas otwierania - sprawdź czujnik		
// Alarm_0226	226	Error	Zacięcie zaworu tłoczenia masy podczas zamykania - sprawdź czujnik		
// Alarm_0227	227	Error	Zacięcie zaworu tłoczenia masy podczas otwierania - sprawdź czujnik		
// Alarm_0228	228	Error	Zacięcie tacki przy otwieraniu - sprawdź czujnik		
// Alarm_0229	229	Error	Zacięcie tacki przy zamykaniu - sprawdź czujnik		
// Alarm_0230	230	Error	Próba uruchomienia z zbyt niską pozycją wylewki względem chwytaka - zmień pozycję gotowości dozownika lub chwytaka		


IF bAlarmInit THEN
    bAlarmInit := FALSE; 
	fbSourceInfo.Clear();
	fbSourceInfo.sName:=wsLiteral_TO_UTF8(sStationName);//'Machine';
	fbSourceInfo.nId:=iStationIndex;//2700;
	// Alarm_0220	220	Error	Błąd napędu tłoka - upewnij się że został dobrze złożony. Błąd NC: {0}	
    arfbAlarm[0].CreateEx(stEventEntry := TC_EVENTS.AlarmClass.Alarm_0220, bWithConfirmation:= FALSE,  ipSourceInfo:= fbSourceInfo); 
	// Alarm_0221	221	Error	Błąd napędu podnośnika. Błąd NC: {0}		
	arfbAlarm[1].CreateEx(stEventEntry := TC_EVENTS.AlarmClass.Alarm_0221, bWithConfirmation:= FALSE,  ipSourceInfo:= fbSourceInfo); 
	// Alarm_0222	222	Error	Nastawa dozy powyżej maksymalnej wartości - zmniejsz ilość dozy		
	arfbAlarm[2].CreateEx(stEventEntry := TC_EVENTS.AlarmClass.Alarm_0222, bWithConfirmation:= FALSE,  ipSourceInfo:= fbSourceInfo); 
	// Alarm_0223	223	Error	Nastawa dozy poniżej minimalnej wartość - zwiększ ilość dozy		
	arfbAlarm[3].CreateEx(stEventEntry := TC_EVENTS.AlarmClass.Alarm_0223, bWithConfirmation:= FALSE,  ipSourceInfo:= fbSourceInfo); 
	// Alarm_0224	224	Error	Zacięcie zaworu zasysania podczas zamykania - sprawdź czujnik		
	arfbAlarm[4].CreateEx(stEventEntry := TC_EVENTS.AlarmClass.Alarm_0224, bWithConfirmation:= FALSE,  ipSourceInfo:= fbSourceInfo); 
	// Alarm_0225	225	Error	Zacięcie zaworu zasysania masy podczas otwierania - sprawdź czujnik		
	arfbAlarm[5].CreateEx(stEventEntry := TC_EVENTS.AlarmClass.Alarm_0225, bWithConfirmation:= FALSE,  ipSourceInfo:= fbSourceInfo); 
	// Alarm_0226	226	Error	Zacięcie zaworu tłoczenia masy podczas zamykania - sprawdź czujnik		
	arfbAlarm[6].CreateEx(stEventEntry := TC_EVENTS.AlarmClass.Alarm_0226, bWithConfirmation:= FALSE,  ipSourceInfo:= fbSourceInfo); 
	// Alarm_0227	227	Error	Zacięcie zaworu tłoczenia masy podczas otwierania - sprawdź czujnik		
	arfbAlarm[7].CreateEx(stEventEntry := TC_EVENTS.AlarmClass.Alarm_0227, bWithConfirmation:= FALSE,  ipSourceInfo:= fbSourceInfo); 
	// Alarm_0228	228	Error	Zacięcie tacki przy otwieraniu - sprawdź czujnik		
	arfbAlarm[8].CreateEx(stEventEntry := TC_EVENTS.AlarmClass.Alarm_0228, bWithConfirmation:= FALSE,  ipSourceInfo:= fbSourceInfo); 
	// Alarm_0229	229	Error	Zacięcie tacki przy zamykaniu - sprawdź czujnik		
	arfbAlarm[9].CreateEx(stEventEntry := TC_EVENTS.AlarmClass.Alarm_0229, bWithConfirmation:= FALSE,  ipSourceInfo:= fbSourceInfo); 
	// Alarm_0230	230	Error	Próba uruchomienia z zbyt niską pozycją wylewki względem chwytaka - zmień pozycję gotowości dozownika lub chwytaka	
	arfbAlarm[10].CreateEx(stEventEntry := TC_EVENTS.AlarmClass.Alarm_0230, bWithConfirmation:= FALSE,  ipSourceInfo:= fbSourceInfo); 
END_IF



//OBSŁUGA BŁĘDÓW DOZOWNIKA Z PODNOŚNIKIEM EPCO

DispencerAxisRef.ReadStatus();

(**Błąd tylko podczas cyklu*)
bErrorOnlyIfCycleOn :=	(eRunningState=E_DispencerState.ePreparingToDose) OR 
						(eRunningState=E_DispencerState.eDosingPh1) OR 
						(eRunningState=E_DispencerState.eDosingPh2) OR 
						(eRunningState=E_DispencerState.eDosingPh3) OR 
						(eRunningState=E_DispencerState.eDosingDone) OR 
						(eRunningState=E_DispencerState.ePulling) OR 
						(eRunningState=E_DispencerState.eSucking) OR 
						(eRunningState=E_DispencerState.eGoingUp) OR 
						(eRunningState=E_DispencerState.eAborting) OR
						(eRunningState=E_DispencerState.eDoseSucking) OR
						(eRunningState=E_DispencerState.eDoseSuckingDone); 
tonEstopDelay			(IN:=bEstop,	PT:=T#5S); //Opóżnienie po EStopie w celu blokoady błędów, powietrze jest później niż Estop a sygnał z czujnika nie pokazuje braku powietrza bo jest odcinany za tym
						
//**********************LISTA BŁĘDÓW******************************
bStateError:= (eState=E_Station.eError) OR (eState=E_Station.eResetting) OR bIgnoreError;

IF bEnable THEN

	IF DispencerAxisRef.Status.Error THEN
		nDispencerError		:= 1;
	ELSIF mcDispencerMoveAbsolute1.Error THEN
		nDispencerError		:= 2;
	ELSIF mcDispencerMoveAbsolute2.Error THEN
		nDispencerError		:= 3;
	ELSIF mcDispencerMoveAbsolute3.Error THEN
		nDispencerError		:= 4;
	ELSE
		nDispencerError		:= 0;	
	END_IF
	
	// Alarm_0220	220	Error	Błąd napędu tłoka - upewnij się że został dobrze złożony. Błąd NC: {0}		
	//Error 1 - BŁĄD SERWA DOZOWNIKA 
	IF (DispencerAxisRef.Status.Error OR mcDispencerMoveAbsolute1.Error
		OR mcDispencerMoveAbsolute2.Error OR mcDispencerMoveAbsolute3.Error) THEN
		sAlarmTest:=F_AxErrMsg(nDispencerServoErrorNr);
		arfbAlarm[0].ipArguments.Clear() .AddString(sAlarmTest);
		IF NOT arfbAlarm[0].bActive THEN
			arfbAlarm[0].Raise(nTimeStamp:=0);
			bManualPullingLatch:=FALSE;
			mcDispencerPower.Override:=100;
			mcDispencerMoveAbsolute1.Execute:=FALSE;
			mcDispencerMoveAbsolute2.Execute:=FALSE;
			mcDispencerMoveAbsolute3.Execute:=FALSE;
			bSuckingValveActuator:=FALSE;
			bDosingValveActuator:=FALSE;	
		END_IF
		ELSE
		IF arfbAlarm[0].bActive AND bReset THEN
			arfbAlarm[0].Clear(nTimeStamp:=0, bResetConfirmation:= FALSE);
		END_IF
		
// 		bManualPullingLatch:=FALSE;
// 		mcDispencerPower.Override:=100;
// 		bError := TRUE;
// 		mcDispencerMoveAbsolute1.Execute:=FALSE;
// 		mcDispencerMoveAbsolute2.Execute:=FALSE;
// 		mcDispencerMoveAbsolute3.Execute:=FALSE;
// 		nErrorNr:=141;
// 		//nErrorNr := nErrorNr+iStationIndex;
// 		nDispencerServoErrorNr:=DispencerAxisRef.Status.ErrorID;
// 		bSuckingValveActuator:=FALSE;
// 		bDosingValveActuator:=FALSE;
// 		sErrorDescription:=CONCAT(INT_TO_STRING(nDispencerError), '-Błąd napędu tłoka - upewnij się że został dobrze złożony. Błąd NC:');
// 		sErrorDescription2:=F_AxErrMsg(nDispencerServoErrorNr);
	END_IF
	
	IF DispencerLifterAxisRef.Status.Error THEN
		nDispencerLifterError	:= 1;
	ELSIF mcLifterPower.Error THEN
		nDispencerLifterError	:= 2;
	ELSIF mcLifterMoveAbsolute.Error THEN
		nDispencerLifterError	:= 3;
	ELSIF mcLifterMoveAbsolute2.Error THEN
		nDispencerLifterError	:= 4;
	ELSIF mcLifterGearIn.Error THEN
		nDispencerLifterError	:= 5;
	ELSIF mcLifterGearOut.Error THEN	
		nDispencerLifterError	:= 6;
	ELSE
		nDispencerLifterError	:= 0;	
	END_IF
	
	// Alarm_0221	221	Error	Błąd napędu podnośnika. Błąd NC: {0}		
	//Error 2 - BŁĄD SERWA PODNOSNIKA DOZOWNIKA
	tonError2(IN:=(bDispencerWithLifter AND (DispencerLifterAxisRef.Status.Error OR mcLifterPower.Error
					OR mcLifterMoveAbsolute.Error OR mcLifterMoveAbsolute2.Error OR mcLifterGearIn.Error OR mcLifterGearOut.Error)), PT:=T#30MS);
	//IF bDispencerWithLifter AND (DispencerLifterAxisRef.Status.Error OR mcLifterPower.Error OR mcLifterMoveAbsolute.Error) AND NOT bStateError THEN
	IF  tonError2.Q THEN
		sAlarmTest:=F_AxErrMsg(nLifterServoErrorNr);
		arfbAlarm[1].ipArguments.Clear() .AddString(sAlarmTest);
		IF NOT arfbAlarm[1].bActive THEN
			arfbAlarm[1].Raise(nTimeStamp:=0);
			bManualPullingLatch:=FALSE;
			mcDispencerPower.Override:=100;
			mcLifterGearIn.Enable:=FALSE;
			mcLifterGearOut.Execute:=TRUE;
			mcLifterPower.Override:=100;
			mcLifterMoveAbsolute.Execute:=FALSE;
			bSuckingValveActuator:=FALSE;
			bDosingValveActuator:=FALSE;
		END_IF
		ELSE
		IF arfbAlarm[1].bActive AND bReset THEN
			arfbAlarm[1].Clear(nTimeStamp:=0, bResetConfirmation:= FALSE);
		END_IF	
// 		bManualPullingLatch:=FALSE;
// 		bSuckingValveActuator:=FALSE;
// 		bDosingValveActuator:=FALSE;
//		mcDispencerPower.Override:=100;
// 		mcLifterGearIn.Enable:=FALSE;
// 		mcLifterGearOut.Execute:=TRUE;
// 		mcLifterPower.Override:=100;
// 		mcLifterMoveAbsolute.Execute:=FALSE;
// 		bError := TRUE;
// 		nErrorNr:=142;
// 		//nErrorNr := nErrorNr+iStationIndex;
// 		nLifterServoErrorNr:=DispencerLifterAxisRef.Status.ErrorID;
// 		sErrorDescription:= CONCAT(INT_TO_STRING(nDispencerLifterError), '-Błąd napędu podnośnika. Błąd NC:');
// 		sErrorDescription2:=F_AxErrMsg(nLifterServoErrorNr);	
	END_IF;
	
	// Alarm_0222	222	Error	Nastawa dozy powyżej maksymalnej wartości - zmniejsz ilość dozy {0}	
	//Error 3 - Nastawa dozy większa niż objętość robocza dozownika
	IF bRun AND eState=E_Station.eReady AND lrDoseVolume>lrRatedDose THEN
		arfbAlarm[2].ipArguments.Clear() .AddLReal(lrDoseVolume);
		IF NOT arfbAlarm[2].bActive THEN
			arfbAlarm[2].Raise(nTimeStamp:=0);
			bManualPullingLatch:=FALSE;
			bSuckingValveActuator:=FALSE;
			bDosingValveActuator:=FALSE;
			mcDispencerPower.Override:=100;
		END_IF
	ELSE	
		IF  arfbAlarm[2].bActive AND bReset THEN
			arfbAlarm[2].Clear(nTimeStamp:=0, bResetConfirmation:= FALSE);
		END_IF

// 		bError := TRUE;
// 		nErrorNr:=143;
		//nErrorNr := nErrorNr+iStationIndex;
// 		sErrorDescription:='Nastawa dozy powyżej maksymalnej wartości - zmniejsz ilość dozy';
// 		sErrorDescription2:=LREAL_TO_STRING(lrDoseVolume);
	END_IF
	
	// Alarm_0223	223	Error	Nastawa dozy poniżej minimalnej wartość - zwiększ ilość dozy
	//Error 4 - Nastawa dozy mniejsza niż objętość robocza dozownika
	IF bRun AND eState=E_Station.eReady AND lrDoseVolume<0 THEN
		arfbAlarm[3].ipArguments.Clear() .AddLReal(lrDoseVolume);
		IF NOT arfbAlarm[3].bActive THEN
			arfbAlarm[3].Raise(nTimeStamp:=0);
			bManualPullingLatch:=FALSE;
			bSuckingValveActuator:=FALSE;
			bDosingValveActuator:=FALSE;
			mcDispencerPower.Override:=100;
		END_IF
	ELSE	
		IF  arfbAlarm[3].bActive AND bReset THEN
			arfbAlarm[3].Clear(nTimeStamp:=0, bResetConfirmation:= FALSE);
		END_IF
// 		bManualPullingLatch:=FALSE;
// 		bSuckingValveActuator:=FALSE;
// 		bDosingValveActuator:=FALSE;
// 		mcDispencerPower.Override:=100;
// 		bError := TRUE;
// 		nErrorNr:=144;
// 		//nErrorNr := nErrorNr+iStationIndex;
// 		sErrorDescription:='Nastawa dozy poniżej minimalnej wartość - zwiększ ilość dozy';
// 		sErrorDescription2:=LREAL_TO_STRING(lrDoseVolume);
	END_IF
	
	// Alarm_0224	224	Error	Zacięcie zaworu zasysania podczas zamykania - sprawdź czujnik	
	//Error 5 - Blokada zaworu ssania przy zamykaniu																					  (*tylko podczas cyklu*)
	tonSuckingValveCloseError(IN:=NOT bSuckingValveClosedSensor AND NOT bSuckingValveActuator AND bErrorOnlyIfCycleOn, PT:=T#1S);
	IF NOT bIgnoreError AND tonSuckingValveCloseError.Q THEN
		IF NOT arfbAlarm[4].bActive THEN
			arfbAlarm[4].Raise(nTimeStamp:=0);
		END_IF
	ELSE	
		IF  arfbAlarm[4].bActive AND bReset THEN
			arfbAlarm[4].Clear(nTimeStamp:=0, bResetConfirmation:= FALSE);
		END_IF

// 		bError := TRUE;
// 		nErrorNr:=145;
// 		//nErrorNr := nErrorNr+iStationIndex;
// 		sErrorDescription:='Zacięcie zaworu zasysania podczas zamykania - sprawdź czujnik';
	END_IF
	
	//Alarm_0225	225	Error	Zacięcie zaworu zasysania masy podczas otwierania - sprawdź czujnik
	//Error 6 - Blokada zaworu ssania przy zamykaniu																				(*tylko podczas cyklu*)
	tonSuckingValveOpenError(IN:=NOT bSuckingValveOpenedSensor AND bSuckingValveActuator AND bErrorOnlyIfCycleOn, PT:=T#1S);
	IF NOT bIgnoreError AND tonSuckingValveOpenError.Q THEN
		IF NOT arfbAlarm[5].bActive THEN
			arfbAlarm[5].Raise(nTimeStamp:=0);
		END_IF
	ELSE	
		IF  arfbAlarm[5].bActive AND bReset THEN
			arfbAlarm[5].Clear(nTimeStamp:=0, bResetConfirmation:= FALSE);
		END_IF
// 		bError := TRUE;
// 		nErrorNr:=146;
// 		//nErrorNr := nErrorNr+iStationIndex;
// 		sErrorDescription:='Zacięcie zaworu zasysania masy podczas otwierania - sprawdź czujnik';
	END_IF
	
	//Alarm_0226	226	Error	Zacięcie zaworu tłoczenia masy podczas zamykania - sprawdź czujnik
	//Error 7 - Blokada zaworu ssania przy zamykaniu																				(*tylko podczas cyklu*)
	tonDosingValveCloseError(IN:=NOT bDosingValveClosedSensor AND NOT bDosingValveActuator AND bErrorOnlyIfCycleOn, PT:=T#1S);
	IF NOT bIgnoreError AND tonDosingValveCloseError.Q THEN
		IF NOT arfbAlarm[6].bActive THEN
			arfbAlarm[6].Raise(nTimeStamp:=0);
		END_IF
	ELSE	
		IF  arfbAlarm[6].bActive AND bReset THEN
			arfbAlarm[6].Clear(nTimeStamp:=0, bResetConfirmation:= FALSE);
		END_IF
// 		bError := TRUE;
// 		nErrorNr:=147;
// 		//nErrorNr := nErrorNr+iStationIndex;
// 		sErrorDescription:='Zacięcie zaworu tłoczenia masy podczas zamykania - sprawdź czujnik';
	END_IF
	
	//Alarm_0227	227	Error	Zacięcie zaworu tłoczenia masy podczas otwierania - sprawdź czujnik
	//Error 8 - Blokada zaworu ssania przy zamykaniu																			  (*tylko podczas cyklu*)
	tonDosingValveOpenError(IN:=NOT bDosingValveOpenedSensor AND bDosingValveActuator AND tonEstopDelay.Q AND NOT bStateError AND bErrorOnlyIfCycleOn, PT:=T#1S);
	IF NOT bIgnoreError AND tonDosingValveOpenError.Q AND NOT bStateError THEN
		IF NOT arfbAlarm[7].bActive THEN
			arfbAlarm[7].Raise(nTimeStamp:=0);
		END_IF
	ELSE	
		IF  arfbAlarm[7].bActive AND bReset THEN
			arfbAlarm[7].Clear(nTimeStamp:=0, bResetConfirmation:= FALSE);
		END_IF
// 		bError := TRUE;
// 		nErrorNr:=148;
// 		//nErrorNr := nErrorNr+iStationIndex;
// 		sErrorDescription:='Zacięcie zaworu tłoczenia masy podczas otwierania - sprawdź czujnik';
	END_IF
	
	//Alarm_0228	228	Error	Zacięcie tacki przy otwieraniu - sprawdź czujnik
	//Error 10 - Blokada tacki przy otwieraniu																 (*tylko podczas cyklu*)
	tonDropCatcherCloseError(IN:=bDropCatcherBackSensor AND bDropCatcherActuator AND  tonEstopDelay.Q AND
		(DispencerLifterAxisRef.NcToPlc.ActPos  >= (lrDropCatcherHeightCV+(lrDropCatcherOpenDistance-5)) AND lrDropCatcherHeightCV>1 AND NOT bHoming AND NOT bHeightSet)
		AND NOT (eDropCatcherState = E_Station.eHoming)
	, PT:=T#13S);
	IF NOT bIgnoreError AND tonDropCatcherCloseError.Q  THEN
		IF NOT arfbAlarm[8].bActive THEN
			arfbAlarm[8].Raise(nTimeStamp:=0);
		END_IF
	ELSE	
		IF  arfbAlarm[8].bActive AND bReset THEN
			arfbAlarm[8].Clear(nTimeStamp:=0, bResetConfirmation:= FALSE);
		END_IF
// 		bError := TRUE;
// 		nErrorNr:=149;
// 		//nErrorNr := nErrorNr+iStationIndex;
// 		sErrorDescription:='Zacięcie tacki przy otwieraniu - sprawdź czujnik';
// 		sErrorDescription2:='';
	END_IF
	
	//Alarm_0229	229	Error	Zacięcie tacki przy zamykaniu - sprawdź czujnik
	//Error 11 - Blokada tacki przy zamykaniu															 (*tylko podczas cyklu*)
	tonDropCatcherOpenError(IN:=NOT bDropCatcherBackSensor AND NOT bDropCatcherActuator AND tonEstopDelay.Q, PT:=T#1S500MS); // było 1S500MS
	IF 	NOT bIgnoreError AND (tonDropCatcherOpenError.Q  OR
        (bRun AND eRunningState>=E_DispencerState.eDosingPh1 AND eRunningState<= E_DispencerState.eDosingPh3 AND NOT bDropCatcherBackSensor)) THEN 
		IF NOT arfbAlarm[9].bActive THEN
			arfbAlarm[9].Raise(nTimeStamp:=0);
		END_IF
	ELSE	
		IF  arfbAlarm[9].bActive AND bReset THEN
			arfbAlarm[9].Clear(nTimeStamp:=0, bResetConfirmation:= FALSE);
		END_IF
// 		bError := TRUE;
// 		nErrorNr:=150;
// 		//nErrorNr := nErrorNr+iStationIndex;
// 		sErrorDescription:='Zacięcie tacki przy zamykaniu - sprawdź czujnik';
// 		sErrorDescription2:='';
	END_IF
	
	//Alarm_0230	230	Error	Próba uruchomienia z zbyt niską pozycją wylewki względem chwytaka - zmień pozycję gotowości dozownika lub chwytaka
	//Error 12 - Próba uruchomienia z zbyt nisko ustawionym chwytakiem (możliwość wylewki w butelce)
	IF NOT bIgnoreError AND 
	(
	(lrLifterActualPosition<(lrDropCatcherHeightCV-40) AND bCatchEnable) OR
	(lrLifterActualPosition<(lrDropCatcherHeightCV-80) AND NOT bCatchEnable) 	
	)
	AND eGlobalState=E_PMLState.ePMLState_STARTING THEN
		IF NOT arfbAlarm[10].bActive THEN
			arfbAlarm[10].Raise(nTimeStamp:=0);
		END_IF
	ELSE	
		IF  arfbAlarm[10].bActive AND bReset THEN
			arfbAlarm[10].Clear(nTimeStamp:=0, bResetConfirmation:= FALSE);
		END_IF
// 		bError := TRUE;
// 		nErrorNr:=151;
// 		//nErrorNr := nErrorNr+iStationIndex;
// 		sErrorDescription:='Próba uruchomienia z zbyt niską pozycją wylewki względem chwytaka - zmień pozycję gotowości dozownika lub chwytaka';
// 		sErrorDescription2:='';
	END_IF	
	
	
ELSE
	bError := FALSE;
END_IF

(*Wyświetlanie błedu na wyjściu*)
bError							:= FALSE;
FOR nAlarmNumerator := 0 TO 19 DO
	bError						:= bError OR arfbAlarm[nAlarmNumerator].bActive;
END_FOR

//Procedura obsługi resetu w zależności od błędu
tofReset(IN:=bReset , PT:=T#3S);
//******************PRZEJŚCIE DO eERROR*****************************

IF bError AND NOT bStateError AND bEStop THEN
	IF eLastState = eRunning THEN
		bCycleNotDone := TRUE;
	END_IF
	eState := E_Station.eError;
END_IF

//****************WYŚWIETLANIE STATUSU BLEDU***********************



(*Wyświetlanie błedu na wyjściu*)
bError;

(*Przepisywanie nazwy stacji*)
sErrorStationName:=WSTRING_TO_STRING(sStationName);
END_ACTION

ACTION HardwareHoming:
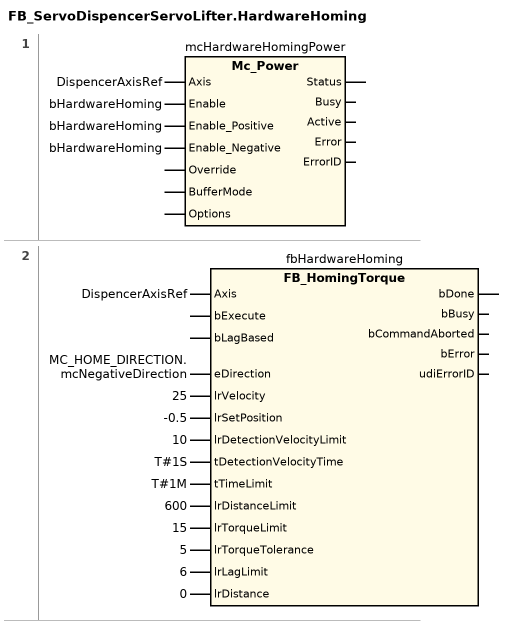
// NETWORK 1
mcHardwareHomingPower(
    Axis := DispencerAxisRef,
    Enable := bHardwareHoming,
    Enable_Positive := bHardwareHoming,
    Enable_Negative := bHardwareHoming); // Mc_Power

// NETWORK 2
fbHardwareHoming(
    Axis := DispencerAxisRef,
    eDirection := MC_HOME_DIRECTION.mcNegativeDirection,
    lrVelocity := 25,
    lrSetPosition := -0.5,
    lrDetectionVelocityLimit := 10,
    tDetectionVelocityTime := T#1S,
    tTimeLimit := T#1M,
    lrDistanceLimit := 600,
    lrTorqueLimit := 15,
    lrTorqueTolerance := 5,
    lrLagLimit := 6,
    lrDistance := 0); // FB_HomingTorque
END_ACTION

ACTION Homing:
bDropCatcherActuator 					:= FALSE;

IF bHoming THEN
	IF bDispencerWithLifter THEN
		mcLifterMoveAbsolute.Acceleration	:=lrLifterAcceleration/15;
		mcLifterMoveAbsolute.Velocity		:=lrLifterVelocity/15;
		mcLifterMoveAbsolute.Position		:=lrMaxPosition;
		IF bDropCatcherBackSensor THEN
			mcLifterMoveAbsolute.Execute		:= TRUE;
		END_IF
		mcLifterPower.Override				:=100;
		IF mcLifterMoveAbsolute.Done THEN
			eState							:= E_Station.eHomingDone;
			mcLifterMoveAbsolute.Execute	:= FALSE;
		END_IF
	ELSE
		IF ABS(DispencerLifterAxisRef.NcToPlc.ActPos-lrMaxPosition)<1 THEN
			eState							:= E_Station.eHomingDone;
			mcLifterMoveAbsolute.Execute	:= FALSE;
		END_IF
	END_IF
ELSIF bHeightSet THEN
	mcLifterManualMove.JogForward:=DispencerLifterAxisRef.NcToPlc.ActPos<=lrLifterReadyPosition AND DispencerLifterAxisRef.NcToPlc.ActPos<=lrMaxPosition;
	mcLifterManualMove.JogBackwards:=DispencerLifterAxisRef.NcToPlc.ActPos>=lrLifterReadyPosition AND DispencerLifterAxisRef.NcToPlc.ActPos>=lrMinPosition;
	IF ABS(DispencerLifterAxisRef.NcToPlc.ActPos-lrLifterReadyPosition)<1 THEN
		mcLifterManualMove.JogForward	:= FALSE;
		mcLifterManualMove.JogBackwards	:= FALSE;
		eState:=E_Station.eHomingDone;
		bHeightSetNotDone					:= TRUE;	
	END_IF
END_IF 
(*
IF NOT bHomingDone THEN
	Lifter_FHPP_CTRL.EnableDrive:=TRUE;
	Lifter_FHPP_CTRL.Stop:=TRUE;
	Lifter_FHPP_CTRL.Halt:=TRUE;
	Lifter_FHPP_CTRL.OPM:=1; 
	IF  Lifter_FHPP_CTRL.Ready THEN
		Lifter_FHPP_CTRL.StartHoming := TRUE;
	END_IF
	IF Lifter_FHPP_CTRL.HomingValid AND tonStartHoming.Q THEN
		Lifter_FHPP_CTRL.StartHoming := FALSE;
		eState:=E_Station.eHomingDone;
	END_IF
ELSE
	lrLifterMaxHeight:=275;
	lrLifterMinHeight:=50;
	Lifter_FHPP_CTRL.JoggingPos:=lrLifterActualPosition<=lrLifterReadyPosition AND lrLifterActualPosition<=lrLifterMaxHeight;
	Lifter_FHPP_CTRL.JoggingNeg:=lrLifterActualPosition>=lrLifterReadyPosition AND lrLifterActualPosition>=lrLifterMinHeight;
	IF ABS(lrLifterActualPosition-lrLifterReadyPosition)<1 THEN
		Lifter_FHPP_CTRL.JoggingPos:=FALSE;
		Lifter_FHPP_CTRL.JoggingNeg:=FALSE;
		eState:=E_Station.eHomingDone;

		
	END_IF		
END_IF*)
END_ACTION

ACTION LifterControlBlocks:
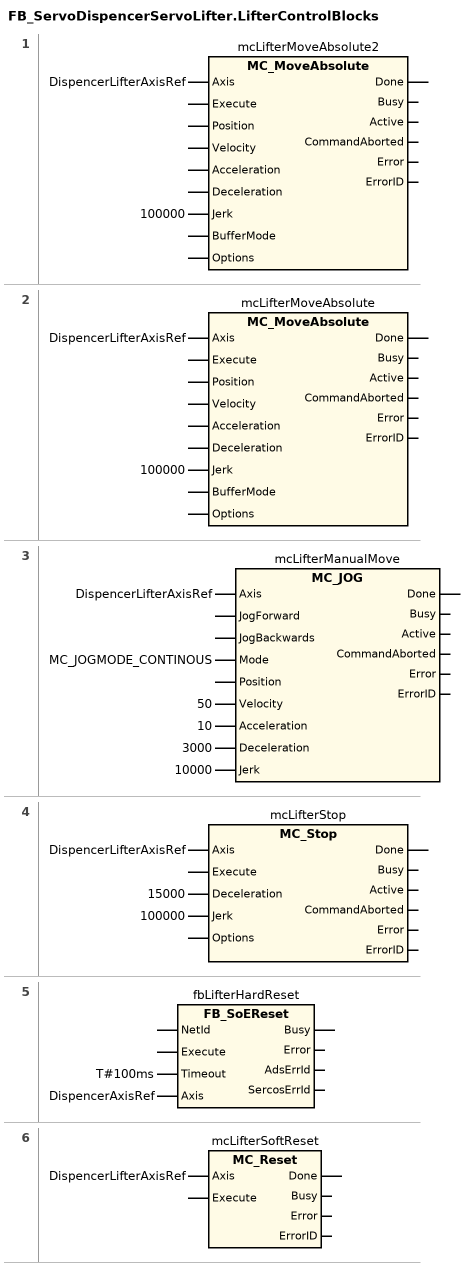
// NETWORK 1
mcLifterMoveAbsolute2(Axis := DispencerLifterAxisRef, Jerk := 100000); // MC_MoveAbsolute

// NETWORK 2
mcLifterMoveAbsolute(Axis := DispencerLifterAxisRef, Jerk := 100000); // MC_MoveAbsolute

// NETWORK 3
mcLifterManualMove(
    Axis := DispencerLifterAxisRef,
    Mode := MC_JOGMODE_CONTINOUS,
    Velocity := 50,
    Acceleration := 10,
    Deceleration := 3000,
    Jerk := 10000); // MC_JOG

// NETWORK 4
mcLifterStop(Axis := DispencerLifterAxisRef, Deceleration := 15000, Jerk := 100000); // MC_Stop

// NETWORK 5
fbLifterHardReset(Timeout := T#100ms, Axis := DispencerAxisRef); // FB_SoEReset

// NETWORK 6
mcLifterSoftReset(Axis := DispencerLifterAxisRef); // MC_Reset

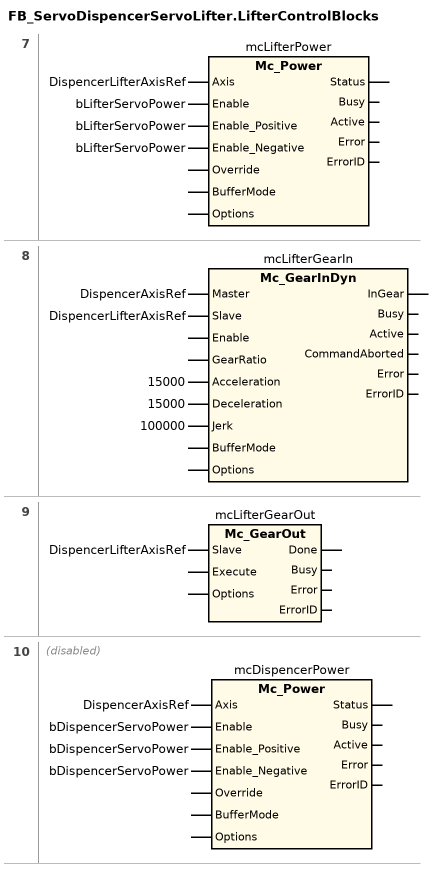
// NETWORK 7
mcLifterPower(
    Axis := DispencerLifterAxisRef,
    Enable := bLifterServoPower,
    Enable_Positive := bLifterServoPower,
    Enable_Negative := bLifterServoPower); // Mc_Power

// NETWORK 8
mcLifterGearIn(
    Master := DispencerAxisRef,
    Slave := DispencerLifterAxisRef,
    Acceleration := 15000,
    Deceleration := 15000,
    Jerk := 100000); // Mc_GearInDyn

// NETWORK 9
mcLifterGearOut(Slave := DispencerLifterAxisRef); // Mc_GearOut

// NETWORK 10 (disabled)
// mcDispencerPower(
//     Axis := DispencerAxisRef,
//     Enable := bDispencerServoPower,
//     Enable_Positive := bDispencerServoPower,
//     Enable_Negative := bDispencerServoPower); // Mc_Power
END_ACTION

ACTION Limits:


(*Prędkość dozowania*)
IF mcDispencerMoveAbsolute1.Velocity	 > lrMaxDispencerVelocity	THEN		mcDispencerMoveAbsolute1.Velocity	:= lrMaxDispencerVelocity;				END_IF
IF mcDispencerMoveAbsolute2.Velocity	 > lrMaxDispencerVelocity	THEN		mcDispencerMoveAbsolute2.Velocity	:= lrMaxDispencerVelocity;				END_IF

(*Pozycja chwytaka DosingDelay*)
IF lrCatchHeightSV < lrLifterStopDosePosition 	THEN		lrCatchHeightSV	:=	lrLifterStopDosePosition;				END_IF
IF lrCatchHeightSV > lrLifterReadyPosition 	  	THEN		lrCatchHeightSV	:=	lrLifterStopDosePosition;				END_IF

IF lrLifterVelocity		< 10		THEN	lrLifterVelocity := 10; 		END_IF
IF lrLifterAcceleration < 100		THEN	lrLifterAcceleration := 100;	END_IF
IF lrLifterDeceleration < 100		THEN	lrLifterDeceleration := 100;	END_IF

(*Doza*)
IF lrDoseVolume			< 10		THEN	lrDoseVolume	:=	10;			END_IF
(*Inny parametr*)
//...
END_ACTION

ACTION ManualMovements:
//W trybie ruchów manualnych wykonuj ruchy za pomocą rozkazów manualnych
IF NOT bDoSmallSucking THEN
	IF NOT bRun AND NOT (eRunningState=E_DispencerState.ePulling) 
				AND NOT (eRunningState=E_DispencerState.eCleaning) 
	THEN
		mcDispencerPower.Override			:=	lrManualOverride;
		mcDispencerManualMove.JogForward	:=	bManualPistonForward;
		mcDispencerManualMove.JogBackwards	:=	bManualPistonBack;
		bSuckingValveActuator				:=	bManualSuckingValve;
		bDosingValveActuator				:=	bManualDosingValve;
		bDropCatcherActuator				:=	bManualDropCatcherForward;
		mcLifterManualMove.JogForward		:=	bManualLifterUp;
		mcLifterManualMove.JogBackwards		:=	bManualLifterDown;
		IF bManualPullingFast OR bManualPullingSlow OR bManualPullingLatch THEN
			bManualPullingLatch				:=	TRUE;
			bDropCatcherActuator			:=	FALSE;
			eRunningState					:=	E_DispencerState.ePulling;
			bManualPullingLatch				:=	FALSE;			
		END_IF	
	ELSE	//Kasuje zeby po cyklu nic sie nie poruszało
		IF NOT (eRunningState=E_DispencerState.ePulling) THEN
			mcDispencerMoveAbsolute1.Execute	:=	FALSE;
		END_IF
		mcDispencerManualMove.JogForward		:=	FALSE;
		mcDispencerManualMove.JogBackwards		:=	FALSE;
	END_IF
END_IF

IF bHoming OR bHeightSet THEN
	eState:=E_Station.eHoming;
END_IF
	
Running();
ManualMovementsStepMode();

